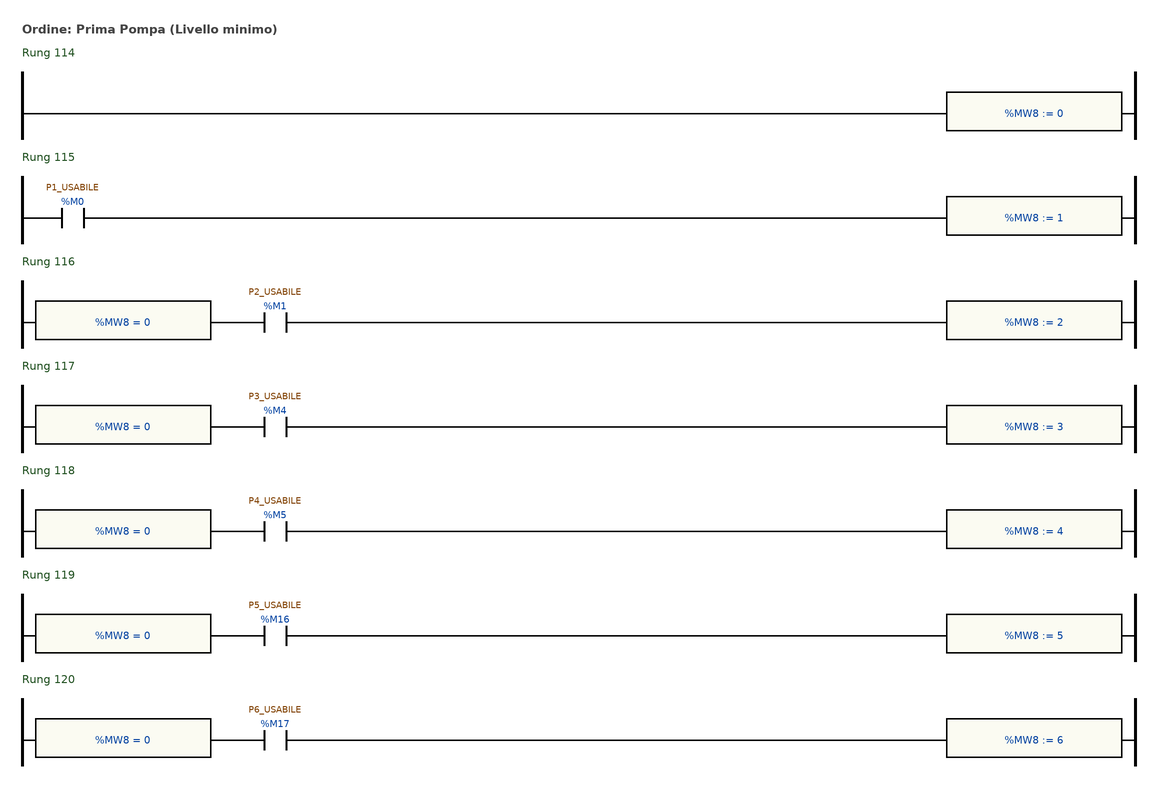

// Rung 114
  LD 1
  [ %MW8 := 0 ]           (* ORDINE_PRIMA_POMPA *)
  // as ST:
  //   ORDINE_PRIMA_POMPA := 0;

// Rung 115
  LD %M0                  (* P1_USABILE *)
  [ %MW8 := 1 ]           (* ORDINE_PRIMA_POMPA *)
  // as ST:
  //   IF P1_USABILE THEN ORDINE_PRIMA_POMPA := 1; END_IF;

// Rung 116
  LD [ %MW8 = 0 ]         (* ORDINE_PRIMA_POMPA *)
  AND %M1                 (* P2_USABILE *)
  [ %MW8 := 2 ]           (* ORDINE_PRIMA_POMPA *)
  // as ST:
  //   IF ORDINE_PRIMA_POMPA = 0 AND P2_USABILE THEN ORDINE_PRIMA_POMPA := 2; END_IF;

// Rung 117
  LD [ %MW8 = 0 ]         (* ORDINE_PRIMA_POMPA *)
  AND %M4                 (* P3_USABILE *)
  [ %MW8 := 3 ]           (* ORDINE_PRIMA_POMPA *)
  // as ST:
  //   IF ORDINE_PRIMA_POMPA = 0 AND P3_USABILE THEN ORDINE_PRIMA_POMPA := 3; END_IF;

// Rung 118
  LD [ %MW8 = 0 ]         (* ORDINE_PRIMA_POMPA *)
  AND %M5                 (* P4_USABILE *)
  [ %MW8 := 4 ]           (* ORDINE_PRIMA_POMPA *)
  // as ST:
  //   IF ORDINE_PRIMA_POMPA = 0 AND P4_USABILE THEN ORDINE_PRIMA_POMPA := 4; END_IF;

// Rung 119
  LD [ %MW8 = 0 ]         (* ORDINE_PRIMA_POMPA *)
  AND %M16                (* P5_USABILE *)
  [ %MW8 := 5 ]           (* ORDINE_PRIMA_POMPA *)
  // as ST:
  //   IF ORDINE_PRIMA_POMPA = 0 AND P5_USABILE THEN ORDINE_PRIMA_POMPA := 5; END_IF;

// Rung 120
  LD [ %MW8 = 0 ]         (* ORDINE_PRIMA_POMPA *)
  AND %M17                (* P6_USABILE *)
  [ %MW8 := 6 ]           (* ORDINE_PRIMA_POMPA *)
  // as ST:
  //   IF ORDINE_PRIMA_POMPA = 0 AND P6_USABILE THEN ORDINE_PRIMA_POMPA := 6; END_IF;

Subroutine Ordine: Seconda Pompa (Livello minimo)
  (* SectionNumber=17, Number=15 *)

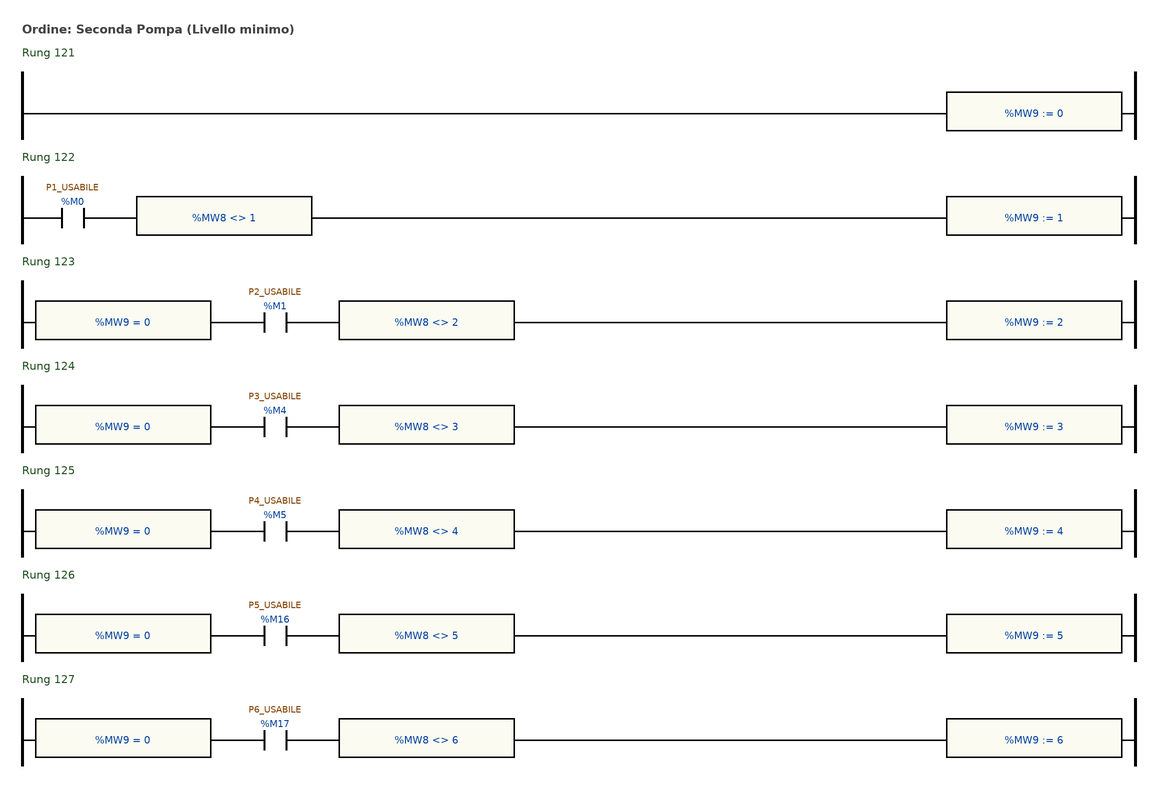

// Rung 121
  LD 1
  [ %MW9 := 0 ]           (* ORDINE_SECONDA_POMPA *)
  // as ST:
  //   ORDINE_SECONDA_POMPA := 0;

// Rung 122
  LD %M0                  (* P1_USABILE *)
  AND [ %MW8 <> 1 ]       (* ORDINE_PRIMA_POMPA *)
  [ %MW9 := 1 ]           (* ORDINE_SECONDA_POMPA *)
  // as ST:
  //   IF P1_USABILE AND ORDINE_PRIMA_POMPA <> 1 THEN ORDINE_SECONDA_POMPA := 1; END_IF;

// Rung 123
  LD [ %MW9 = 0 ]         (* ORDINE_SECONDA_POMPA *)
  AND %M1                 (* P2_USABILE *)
  AND [ %MW8 <> 2 ]       (* ORDINE_PRIMA_POMPA *)
  [ %MW9 := 2 ]           (* ORDINE_SECONDA_POMPA *)
  // as ST:
  //   IF ORDINE_SECONDA_POMPA = 0 AND P2_USABILE AND ORDINE_PRIMA_POMPA <> 2 THEN ORDINE_SECONDA_POMPA := 2; END_IF;

// Rung 124
  LD [ %MW9 = 0 ]         (* ORDINE_SECONDA_POMPA *)
  AND %M4                 (* P3_USABILE *)
  AND [ %MW8 <> 3 ]       (* ORDINE_PRIMA_POMPA *)
  [ %MW9 := 3 ]           (* ORDINE_SECONDA_POMPA *)
  // as ST:
  //   IF ORDINE_SECONDA_POMPA = 0 AND P3_USABILE AND ORDINE_PRIMA_POMPA <> 3 THEN ORDINE_SECONDA_POMPA := 3; END_IF;

// Rung 125
  LD [ %MW9 = 0 ]         (* ORDINE_SECONDA_POMPA *)
  AND %M5                 (* P4_USABILE *)
  AND [ %MW8 <> 4 ]       (* ORDINE_PRIMA_POMPA *)
  [ %MW9 := 4 ]           (* ORDINE_SECONDA_POMPA *)
  // as ST:
  //   IF ORDINE_SECONDA_POMPA = 0 AND P4_USABILE AND ORDINE_PRIMA_POMPA <> 4 THEN ORDINE_SECONDA_POMPA := 4; END_IF;

// Rung 126
  LD [ %MW9 = 0 ]         (* ORDINE_SECONDA_POMPA *)
  AND %M16                (* P5_USABILE *)
  AND [ %MW8 <> 5 ]       (* ORDINE_PRIMA_POMPA *)
  [ %MW9 := 5 ]           (* ORDINE_SECONDA_POMPA *)
  // as ST:
  //   IF ORDINE_SECONDA_POMPA = 0 AND P5_USABILE AND ORDINE_PRIMA_POMPA <> 5 THEN ORDINE_SECONDA_POMPA := 5; END_IF;

// Rung 127
  LD [ %MW9 = 0 ]         (* ORDINE_SECONDA_POMPA *)
  AND %M17                (* P6_USABILE *)
  AND [ %MW8 <> 6 ]       (* ORDINE_PRIMA_POMPA *)
  [ %MW9 := 6 ]           (* ORDINE_SECONDA_POMPA *)
  // as ST:
  //   IF ORDINE_SECONDA_POMPA = 0 AND P6_USABILE AND ORDINE_PRIMA_POMPA <> 6 THEN ORDINE_SECONDA_POMPA := 6; END_IF;

Subroutine Comanda: Prima Pompa (Livello minimo)
  (* SectionNumber=18, Number=16 *)

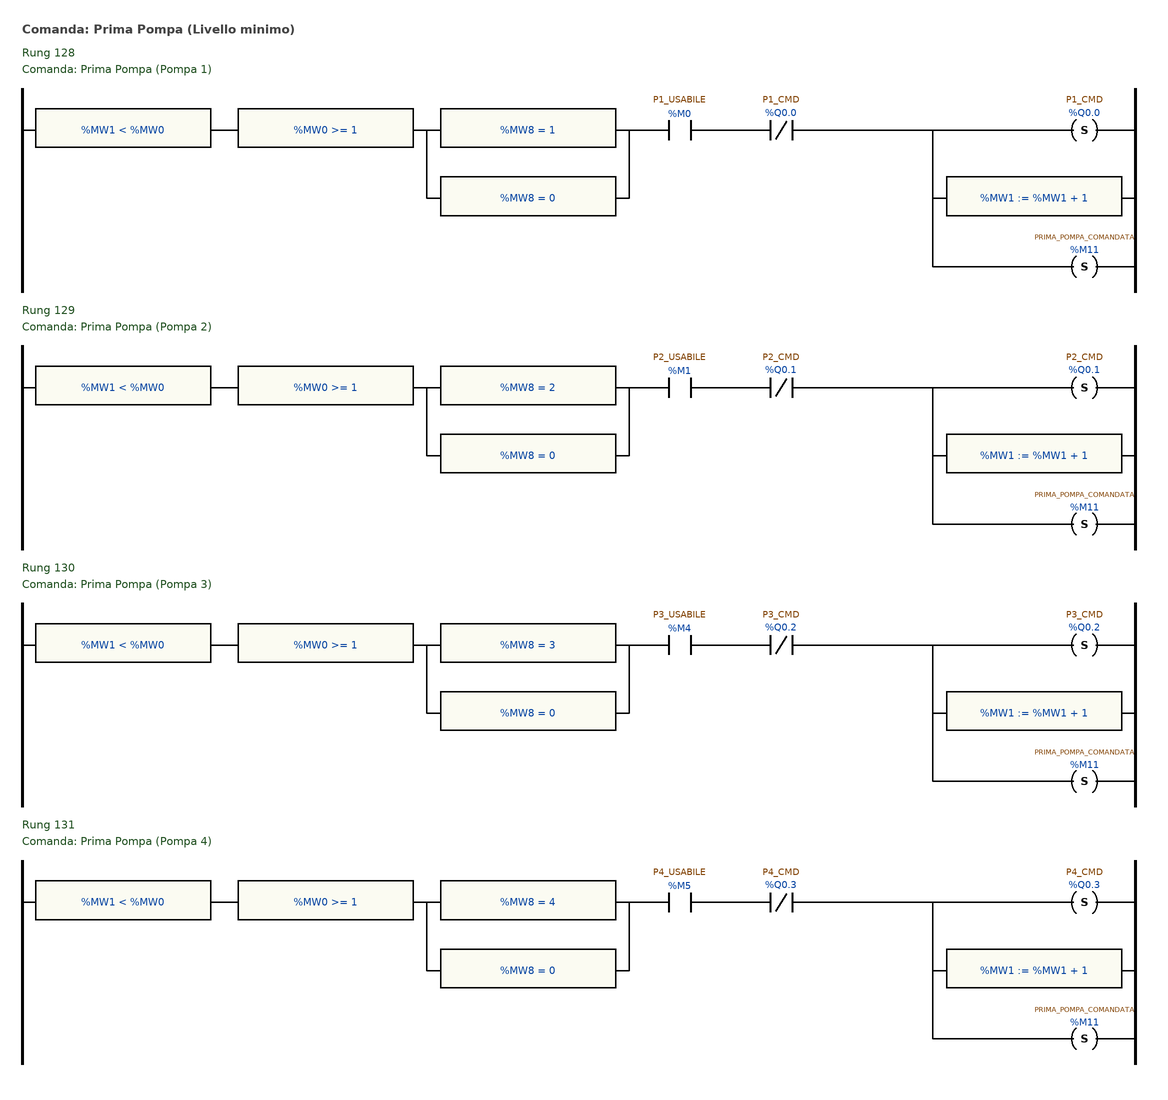

// Rung 128
// Comanda: Prima Pompa (Pompa 1)
  LD [ %MW1 < %MW0 ]      (* NUM_POMPE_COMANDATE, NUM_POMPE_DA_COMANDARE *)
  AND [ %MW0 >= 1 ]       (* NUM_POMPE_DA_COMANDARE *)
  AND( [ %MW8 = 1 ]       (* ORDINE_PRIMA_POMPA *)
  OR [ %MW8 = 0 ]         (* ORDINE_PRIMA_POMPA *)
  )
  AND %M0                 (* P1_USABILE *)
  ANDN %Q0.0              (* P1_CMD *)
  S %Q0.0                 (* P1_CMD *)
  [ %MW1 := %MW1 + 1 ]    (* NUM_POMPE_COMANDATE, NUM_POMPE_COMANDATE *)
  S %M11                  (* PRIMA_POMPA_COMANDATA *)
  // as ST:
  //   _t1 := NUM_POMPE_COMANDATE < NUM_POMPE_DA_COMANDARE AND NUM_POMPE_DA_COMANDARE >= 1 AND (ORDINE_PRIMA_POMPA = 1 OR ORDINE_PRIMA_POMPA = 0) AND P1_USABILE AND NOT P1_CMD;
  //   IF _t1 THEN P1_CMD := TRUE; END_IF;
  //   IF _t1 THEN NUM_POMPE_COMANDATE := NUM_POMPE_COMANDATE + 1; END_IF;
  //   IF _t1 THEN PRIMA_POMPA_COMANDATA := TRUE; END_IF;

// Rung 129
// Comanda: Prima Pompa (Pompa 2)
  LD [ %MW1 < %MW0 ]      (* NUM_POMPE_COMANDATE, NUM_POMPE_DA_COMANDARE *)
  AND [ %MW0 >= 1 ]       (* NUM_POMPE_DA_COMANDARE *)
  AND( [ %MW8 = 2 ]       (* ORDINE_PRIMA_POMPA *)
  OR [ %MW8 = 0 ]         (* ORDINE_PRIMA_POMPA *)
  )
  AND %M1                 (* P2_USABILE *)
  ANDN %Q0.1              (* P2_CMD *)
  S %Q0.1                 (* P2_CMD *)
  [ %MW1 := %MW1 + 1 ]    (* NUM_POMPE_COMANDATE, NUM_POMPE_COMANDATE *)
  S %M11                  (* PRIMA_POMPA_COMANDATA *)
  // as ST:
  //   _t1 := NUM_POMPE_COMANDATE < NUM_POMPE_DA_COMANDARE AND NUM_POMPE_DA_COMANDARE >= 1 AND (ORDINE_PRIMA_POMPA = 2 OR ORDINE_PRIMA_POMPA = 0) AND P2_USABILE AND NOT P2_CMD;
  //   IF _t1 THEN P2_CMD := TRUE; END_IF;
  //   IF _t1 THEN NUM_POMPE_COMANDATE := NUM_POMPE_COMANDATE + 1; END_IF;
  //   IF _t1 THEN PRIMA_POMPA_COMANDATA := TRUE; END_IF;

// Rung 130
// Comanda: Prima Pompa (Pompa 3)
  LD [ %MW1 < %MW0 ]      (* NUM_POMPE_COMANDATE, NUM_POMPE_DA_COMANDARE *)
  AND [ %MW0 >= 1 ]       (* NUM_POMPE_DA_COMANDARE *)
  AND( [ %MW8 = 3 ]       (* ORDINE_PRIMA_POMPA *)
  OR [ %MW8 = 0 ]         (* ORDINE_PRIMA_POMPA *)
  )
  AND %M4                 (* P3_USABILE *)
  ANDN %Q0.2              (* P3_CMD *)
  S %Q0.2                 (* P3_CMD *)
  [ %MW1 := %MW1 + 1 ]    (* NUM_POMPE_COMANDATE, NUM_POMPE_COMANDATE *)
  S %M11                  (* PRIMA_POMPA_COMANDATA *)
  // as ST:
  //   _t1 := NUM_POMPE_COMANDATE < NUM_POMPE_DA_COMANDARE AND NUM_POMPE_DA_COMANDARE >= 1 AND (ORDINE_PRIMA_POMPA = 3 OR ORDINE_PRIMA_POMPA = 0) AND P3_USABILE AND NOT P3_CMD;
  //   IF _t1 THEN P3_CMD := TRUE; END_IF;
  //   IF _t1 THEN NUM_POMPE_COMANDATE := NUM_POMPE_COMANDATE + 1; END_IF;
  //   IF _t1 THEN PRIMA_POMPA_COMANDATA := TRUE; END_IF;

// Rung 131
// Comanda: Prima Pompa (Pompa 4)
  LD [ %MW1 < %MW0 ]      (* NUM_POMPE_COMANDATE, NUM_POMPE_DA_COMANDARE *)
  AND [ %MW0 >= 1 ]       (* NUM_POMPE_DA_COMANDARE *)
  AND( [ %MW8 = 4 ]       (* ORDINE_PRIMA_POMPA *)
  OR [ %MW8 = 0 ]         (* ORDINE_PRIMA_POMPA *)
  )
  AND %M5                 (* P4_USABILE *)
  ANDN %Q0.3              (* P4_CMD *)
  S %Q0.3                 (* P4_CMD *)
  [ %MW1 := %MW1 + 1 ]    (* NUM_POMPE_COMANDATE, NUM_POMPE_COMANDATE *)
  S %M11                  (* PRIMA_POMPA_COMANDATA *)
  // as ST:
  //   _t1 := NUM_POMPE_COMANDATE < NUM_POMPE_DA_COMANDARE AND NUM_POMPE_DA_COMANDARE >= 1 AND (ORDINE_PRIMA_POMPA = 4 OR ORDINE_PRIMA_POMPA = 0) AND P4_USABILE AND NOT P4_CMD;
  //   IF _t1 THEN P4_CMD := TRUE; END_IF;
  //   IF _t1 THEN NUM_POMPE_COMANDATE := NUM_POMPE_COMANDATE + 1; END_IF;
  //   IF _t1 THEN PRIMA_POMPA_COMANDATA := TRUE; END_IF;

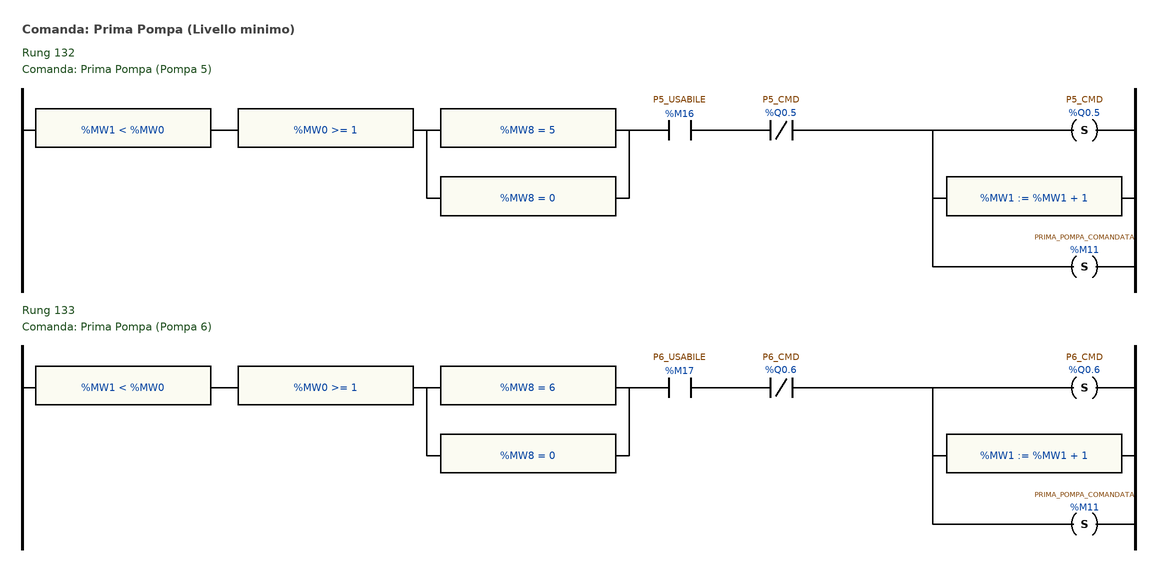

// Rung 132
// Comanda: Prima Pompa (Pompa 5)
  LD [ %MW1 < %MW0 ]      (* NUM_POMPE_COMANDATE, NUM_POMPE_DA_COMANDARE *)
  AND [ %MW0 >= 1 ]       (* NUM_POMPE_DA_COMANDARE *)
  AND( [ %MW8 = 5 ]       (* ORDINE_PRIMA_POMPA *)
  OR [ %MW8 = 0 ]         (* ORDINE_PRIMA_POMPA *)
  )
  AND %M16                (* P5_USABILE *)
  ANDN %Q0.5              (* P5_CMD *)
  S %Q0.5                 (* P5_CMD *)
  [ %MW1 := %MW1 + 1 ]    (* NUM_POMPE_COMANDATE, NUM_POMPE_COMANDATE *)
  S %M11                  (* PRIMA_POMPA_COMANDATA *)
  // as ST:
  //   _t1 := NUM_POMPE_COMANDATE < NUM_POMPE_DA_COMANDARE AND NUM_POMPE_DA_COMANDARE >= 1 AND (ORDINE_PRIMA_POMPA = 5 OR ORDINE_PRIMA_POMPA = 0) AND P5_USABILE AND NOT P5_CMD;
  //   IF _t1 THEN P5_CMD := TRUE; END_IF;
  //   IF _t1 THEN NUM_POMPE_COMANDATE := NUM_POMPE_COMANDATE + 1; END_IF;
  //   IF _t1 THEN PRIMA_POMPA_COMANDATA := TRUE; END_IF;

// Rung 133
// Comanda: Prima Pompa (Pompa 6)
  LD [ %MW1 < %MW0 ]      (* NUM_POMPE_COMANDATE, NUM_POMPE_DA_COMANDARE *)
  AND [ %MW0 >= 1 ]       (* NUM_POMPE_DA_COMANDARE *)
  AND( [ %MW8 = 6 ]       (* ORDINE_PRIMA_POMPA *)
  OR [ %MW8 = 0 ]         (* ORDINE_PRIMA_POMPA *)
  )
  AND %M17                (* P6_USABILE *)
  ANDN %Q0.6              (* P6_CMD *)
  S %Q0.6                 (* P6_CMD *)
  [ %MW1 := %MW1 + 1 ]    (* NUM_POMPE_COMANDATE, NUM_POMPE_COMANDATE *)
  S %M11                  (* PRIMA_POMPA_COMANDATA *)
  // as ST:
  //   _t1 := NUM_POMPE_COMANDATE < NUM_POMPE_DA_COMANDARE AND NUM_POMPE_DA_COMANDARE >= 1 AND (ORDINE_PRIMA_POMPA = 6 OR ORDINE_PRIMA_POMPA = 0) AND P6_USABILE AND NOT P6_CMD;
  //   IF _t1 THEN P6_CMD := TRUE; END_IF;
  //   IF _t1 THEN NUM_POMPE_COMANDATE := NUM_POMPE_COMANDATE + 1; END_IF;
  //   IF _t1 THEN PRIMA_POMPA_COMANDATA := TRUE; END_IF;

Subroutine Comanda: Seconda Pompa (Livello minimo)
  (* SectionNumber=19, Number=17 *)

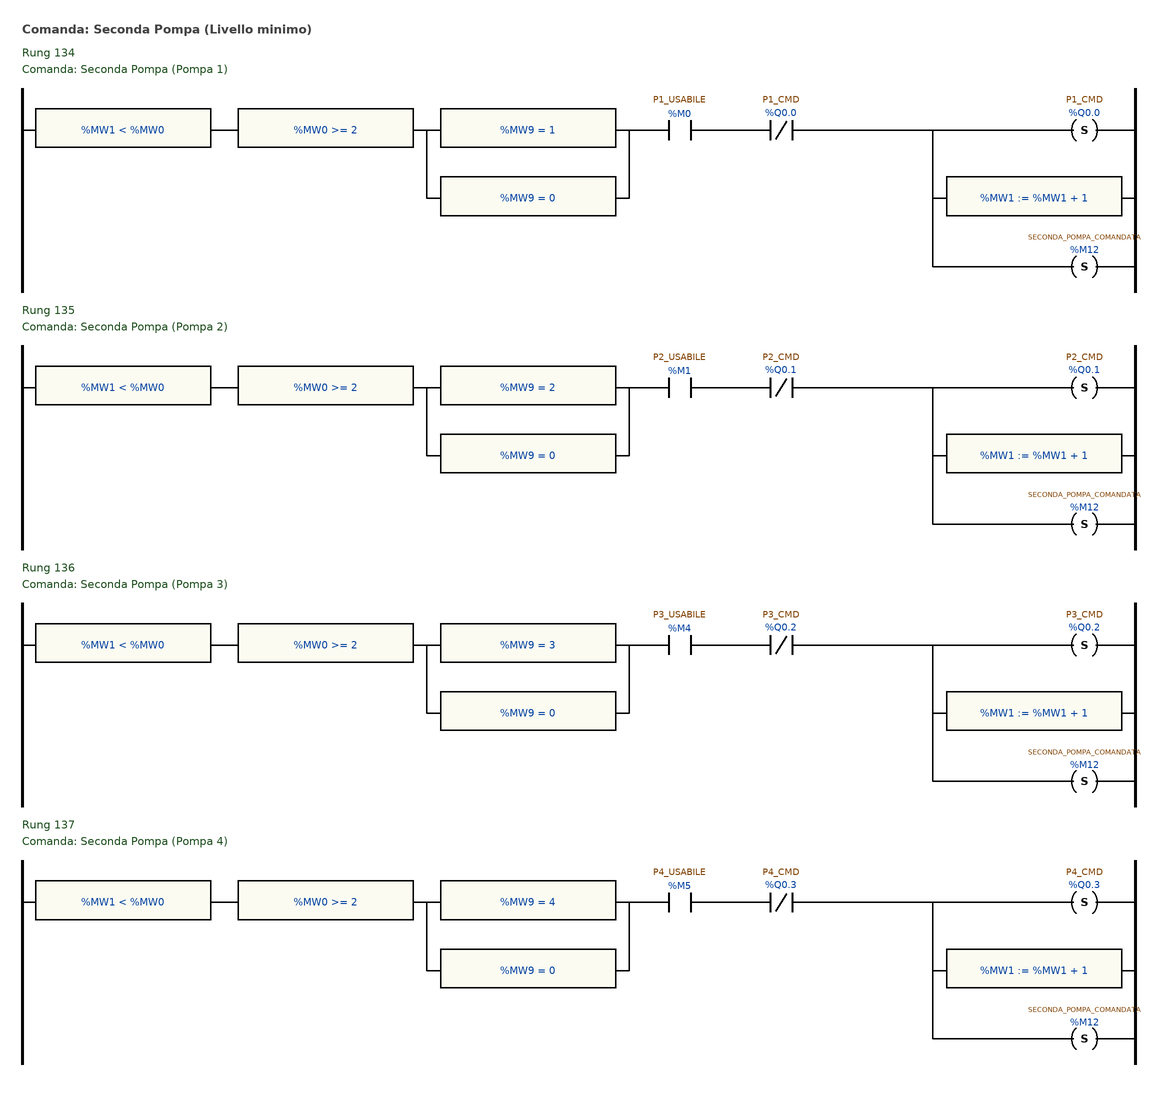

// Rung 134
// Comanda: Seconda Pompa (Pompa 1)
  LD [ %MW1 < %MW0 ]      (* NUM_POMPE_COMANDATE, NUM_POMPE_DA_COMANDARE *)
  AND [ %MW0 >= 2 ]       (* NUM_POMPE_DA_COMANDARE *)
  AND( [ %MW9 = 1 ]       (* ORDINE_SECONDA_POMPA *)
  OR [ %MW9 = 0 ]         (* ORDINE_SECONDA_POMPA *)
  )
  AND %M0                 (* P1_USABILE *)
  ANDN %Q0.0              (* P1_CMD *)
  S %Q0.0                 (* P1_CMD *)
  [ %MW1 := %MW1 + 1 ]    (* NUM_POMPE_COMANDATE, NUM_POMPE_COMANDATE *)
  S %M12                  (* SECONDA_POMPA_COMANDATA *)
  // as ST:
  //   _t1 := NUM_POMPE_COMANDATE < NUM_POMPE_DA_COMANDARE AND NUM_POMPE_DA_COMANDARE >= 2 AND (ORDINE_SECONDA_POMPA = 1 OR ORDINE_SECONDA_POMPA = 0) AND P1_USABILE AND NOT P1_CMD;
  //   IF _t1 THEN P1_CMD := TRUE; END_IF;
  //   IF _t1 THEN NUM_POMPE_COMANDATE := NUM_POMPE_COMANDATE + 1; END_IF;
  //   IF _t1 THEN SECONDA_POMPA_COMANDATA := TRUE; END_IF;

// Rung 135
// Comanda: Seconda Pompa (Pompa 2)
  LD [ %MW1 < %MW0 ]      (* NUM_POMPE_COMANDATE, NUM_POMPE_DA_COMANDARE *)
  AND [ %MW0 >= 2 ]       (* NUM_POMPE_DA_COMANDARE *)
  AND( [ %MW9 = 2 ]       (* ORDINE_SECONDA_POMPA *)
  OR [ %MW9 = 0 ]         (* ORDINE_SECONDA_POMPA *)
  )
  AND %M1                 (* P2_USABILE *)
  ANDN %Q0.1              (* P2_CMD *)
  S %Q0.1                 (* P2_CMD *)
  [ %MW1 := %MW1 + 1 ]    (* NUM_POMPE_COMANDATE, NUM_POMPE_COMANDATE *)
  S %M12                  (* SECONDA_POMPA_COMANDATA *)
  // as ST:
  //   _t1 := NUM_POMPE_COMANDATE < NUM_POMPE_DA_COMANDARE AND NUM_POMPE_DA_COMANDARE >= 2 AND (ORDINE_SECONDA_POMPA = 2 OR ORDINE_SECONDA_POMPA = 0) AND P2_USABILE AND NOT P2_CMD;
  //   IF _t1 THEN P2_CMD := TRUE; END_IF;
  //   IF _t1 THEN NUM_POMPE_COMANDATE := NUM_POMPE_COMANDATE + 1; END_IF;
  //   IF _t1 THEN SECONDA_POMPA_COMANDATA := TRUE; END_IF;

// Rung 136
// Comanda: Seconda Pompa (Pompa 3)
  LD [ %MW1 < %MW0 ]      (* NUM_POMPE_COMANDATE, NUM_POMPE_DA_COMANDARE *)
  AND [ %MW0 >= 2 ]       (* NUM_POMPE_DA_COMANDARE *)
  AND( [ %MW9 = 3 ]       (* ORDINE_SECONDA_POMPA *)
  OR [ %MW9 = 0 ]         (* ORDINE_SECONDA_POMPA *)
  )
  AND %M4                 (* P3_USABILE *)
  ANDN %Q0.2              (* P3_CMD *)
  S %Q0.2                 (* P3_CMD *)
  [ %MW1 := %MW1 + 1 ]    (* NUM_POMPE_COMANDATE, NUM_POMPE_COMANDATE *)
  S %M12                  (* SECONDA_POMPA_COMANDATA *)
  // as ST:
  //   _t1 := NUM_POMPE_COMANDATE < NUM_POMPE_DA_COMANDARE AND NUM_POMPE_DA_COMANDARE >= 2 AND (ORDINE_SECONDA_POMPA = 3 OR ORDINE_SECONDA_POMPA = 0) AND P3_USABILE AND NOT P3_CMD;
  //   IF _t1 THEN P3_CMD := TRUE; END_IF;
  //   IF _t1 THEN NUM_POMPE_COMANDATE := NUM_POMPE_COMANDATE + 1; END_IF;
  //   IF _t1 THEN SECONDA_POMPA_COMANDATA := TRUE; END_IF;

// Rung 137
// Comanda: Seconda Pompa (Pompa 4)
  LD [ %MW1 < %MW0 ]      (* NUM_POMPE_COMANDATE, NUM_POMPE_DA_COMANDARE *)
  AND [ %MW0 >= 2 ]       (* NUM_POMPE_DA_COMANDARE *)
  AND( [ %MW9 = 4 ]       (* ORDINE_SECONDA_POMPA *)
  OR [ %MW9 = 0 ]         (* ORDINE_SECONDA_POMPA *)
  )
  AND %M5                 (* P4_USABILE *)
  ANDN %Q0.3              (* P4_CMD *)
  S %Q0.3                 (* P4_CMD *)
  [ %MW1 := %MW1 + 1 ]    (* NUM_POMPE_COMANDATE, NUM_POMPE_COMANDATE *)
  S %M12                  (* SECONDA_POMPA_COMANDATA *)
  // as ST:
  //   _t1 := NUM_POMPE_COMANDATE < NUM_POMPE_DA_COMANDARE AND NUM_POMPE_DA_COMANDARE >= 2 AND (ORDINE_SECONDA_POMPA = 4 OR ORDINE_SECONDA_POMPA = 0) AND P4_USABILE AND NOT P4_CMD;
  //   IF _t1 THEN P4_CMD := TRUE; END_IF;
  //   IF _t1 THEN NUM_POMPE_COMANDATE := NUM_POMPE_COMANDATE + 1; END_IF;
  //   IF _t1 THEN SECONDA_POMPA_COMANDATA := TRUE; END_IF;

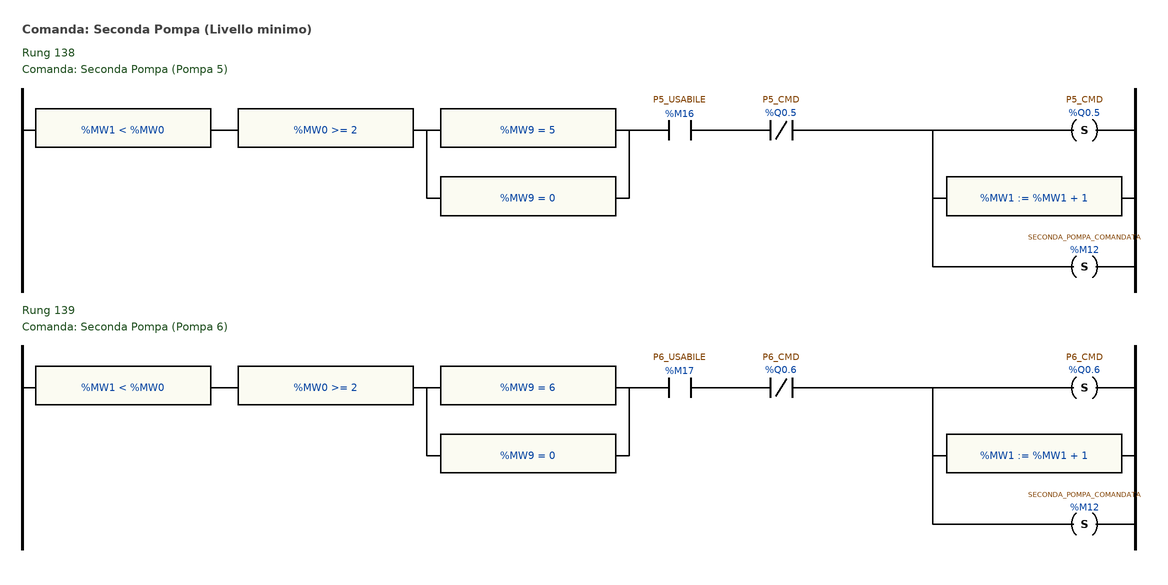

// Rung 138
// Comanda: Seconda Pompa (Pompa 5)
  LD [ %MW1 < %MW0 ]      (* NUM_POMPE_COMANDATE, NUM_POMPE_DA_COMANDARE *)
  AND [ %MW0 >= 2 ]       (* NUM_POMPE_DA_COMANDARE *)
  AND( [ %MW9 = 5 ]       (* ORDINE_SECONDA_POMPA *)
  OR [ %MW9 = 0 ]         (* ORDINE_SECONDA_POMPA *)
  )
  AND %M16                (* P5_USABILE *)
  ANDN %Q0.5              (* P5_CMD *)
  S %Q0.5                 (* P5_CMD *)
  [ %MW1 := %MW1 + 1 ]    (* NUM_POMPE_COMANDATE, NUM_POMPE_COMANDATE *)
  S %M12                  (* SECONDA_POMPA_COMANDATA *)
  // as ST:
  //   _t1 := NUM_POMPE_COMANDATE < NUM_POMPE_DA_COMANDARE AND NUM_POMPE_DA_COMANDARE >= 2 AND (ORDINE_SECONDA_POMPA = 5 OR ORDINE_SECONDA_POMPA = 0) AND P5_USABILE AND NOT P5_CMD;
  //   IF _t1 THEN P5_CMD := TRUE; END_IF;
  //   IF _t1 THEN NUM_POMPE_COMANDATE := NUM_POMPE_COMANDATE + 1; END_IF;
  //   IF _t1 THEN SECONDA_POMPA_COMANDATA := TRUE; END_IF;

// Rung 139
// Comanda: Seconda Pompa (Pompa 6)
  LD [ %MW1 < %MW0 ]      (* NUM_POMPE_COMANDATE, NUM_POMPE_DA_COMANDARE *)
  AND [ %MW0 >= 2 ]       (* NUM_POMPE_DA_COMANDARE *)
  AND( [ %MW9 = 6 ]       (* ORDINE_SECONDA_POMPA *)
  OR [ %MW9 = 0 ]         (* ORDINE_SECONDA_POMPA *)
  )
  AND %M17                (* P6_USABILE *)
  ANDN %Q0.6              (* P6_CMD *)
  S %Q0.6                 (* P6_CMD *)
  [ %MW1 := %MW1 + 1 ]    (* NUM_POMPE_COMANDATE, NUM_POMPE_COMANDATE *)
  S %M12                  (* SECONDA_POMPA_COMANDATA *)
  // as ST:
  //   _t1 := NUM_POMPE_COMANDATE < NUM_POMPE_DA_COMANDARE AND NUM_POMPE_DA_COMANDARE >= 2 AND (ORDINE_SECONDA_POMPA = 6 OR ORDINE_SECONDA_POMPA = 0) AND P6_USABILE AND NOT P6_CMD;
  //   IF _t1 THEN P6_CMD := TRUE; END_IF;
  //   IF _t1 THEN NUM_POMPE_COMANDATE := NUM_POMPE_COMANDATE + 1; END_IF;
  //   IF _t1 THEN SECONDA_POMPA_COMANDATA := TRUE; END_IF;

Subroutine Disattivazione Pompe (Livello minimo)
  (* SectionNumber=20, Number=18 *)

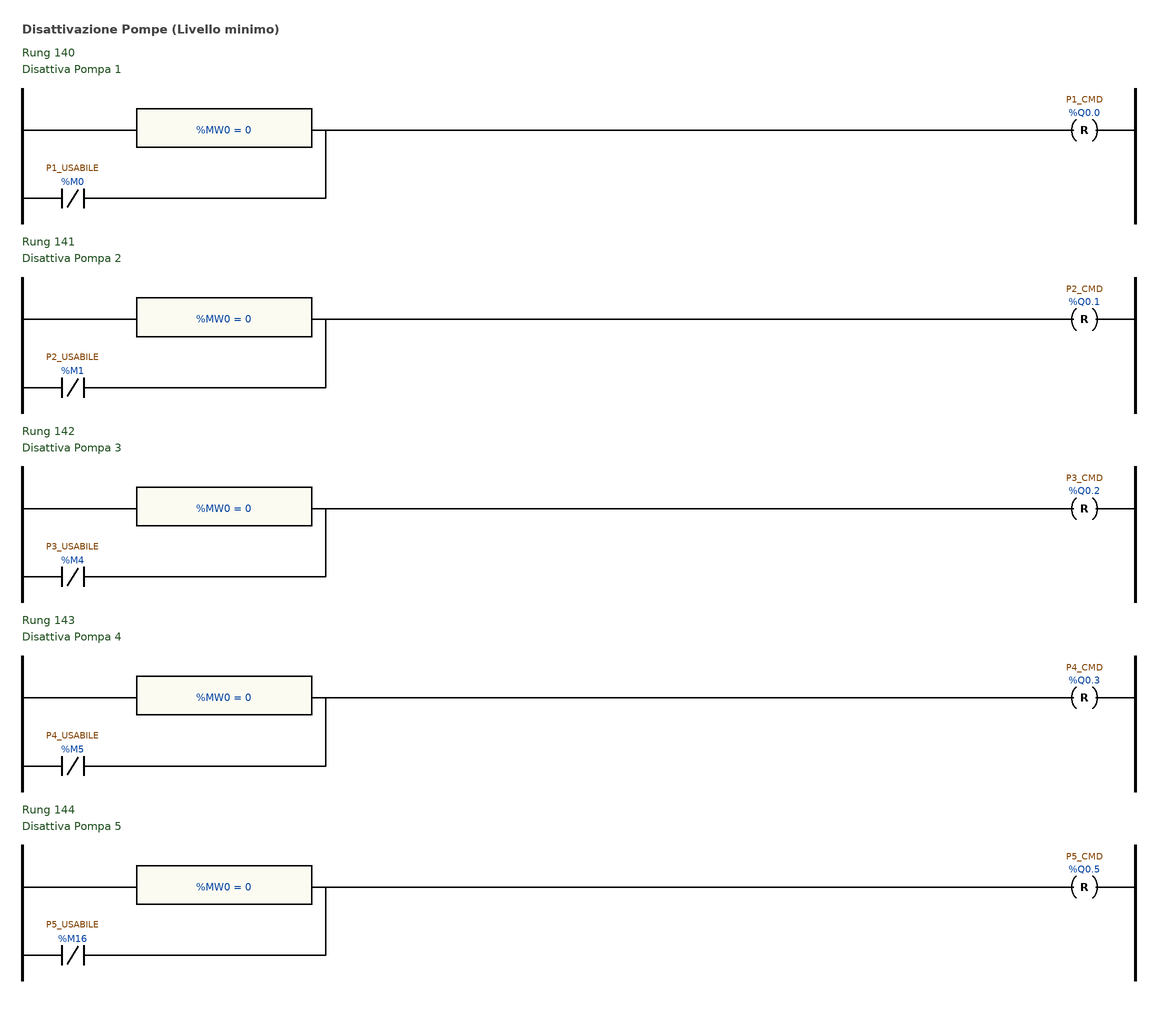

// Rung 140
// Disattiva Pompa 1
  LD [ %MW0 = 0 ]         (* NUM_POMPE_DA_COMANDARE *)
  ORN %M0                 (* P1_USABILE *)
  R %Q0.0                 (* P1_CMD *)
  // as ST:
  //   IF NUM_POMPE_DA_COMANDARE = 0 OR NOT P1_USABILE THEN P1_CMD := FALSE; END_IF;

// Rung 141
// Disattiva Pompa 2
  LD [ %MW0 = 0 ]         (* NUM_POMPE_DA_COMANDARE *)
  ORN %M1                 (* P2_USABILE *)
  R %Q0.1                 (* P2_CMD *)
  // as ST:
  //   IF NUM_POMPE_DA_COMANDARE = 0 OR NOT P2_USABILE THEN P2_CMD := FALSE; END_IF;

// Rung 142
// Disattiva Pompa 3
  LD [ %MW0 = 0 ]         (* NUM_POMPE_DA_COMANDARE *)
  ORN %M4                 (* P3_USABILE *)
  R %Q0.2                 (* P3_CMD *)
  // as ST:
  //   IF NUM_POMPE_DA_COMANDARE = 0 OR NOT P3_USABILE THEN P3_CMD := FALSE; END_IF;

// Rung 143
// Disattiva Pompa 4
  LD [ %MW0 = 0 ]         (* NUM_POMPE_DA_COMANDARE *)
  ORN %M5                 (* P4_USABILE *)
  R %Q0.3                 (* P4_CMD *)
  // as ST:
  //   IF NUM_POMPE_DA_COMANDARE = 0 OR NOT P4_USABILE THEN P4_CMD := FALSE; END_IF;

// Rung 144
// Disattiva Pompa 5
  LD [ %MW0 = 0 ]         (* NUM_POMPE_DA_COMANDARE *)
  ORN %M16                (* P5_USABILE *)
  R %Q0.5                 (* P5_CMD *)
  // as ST:
  //   IF NUM_POMPE_DA_COMANDARE = 0 OR NOT P5_USABILE THEN P5_CMD := FALSE; END_IF;

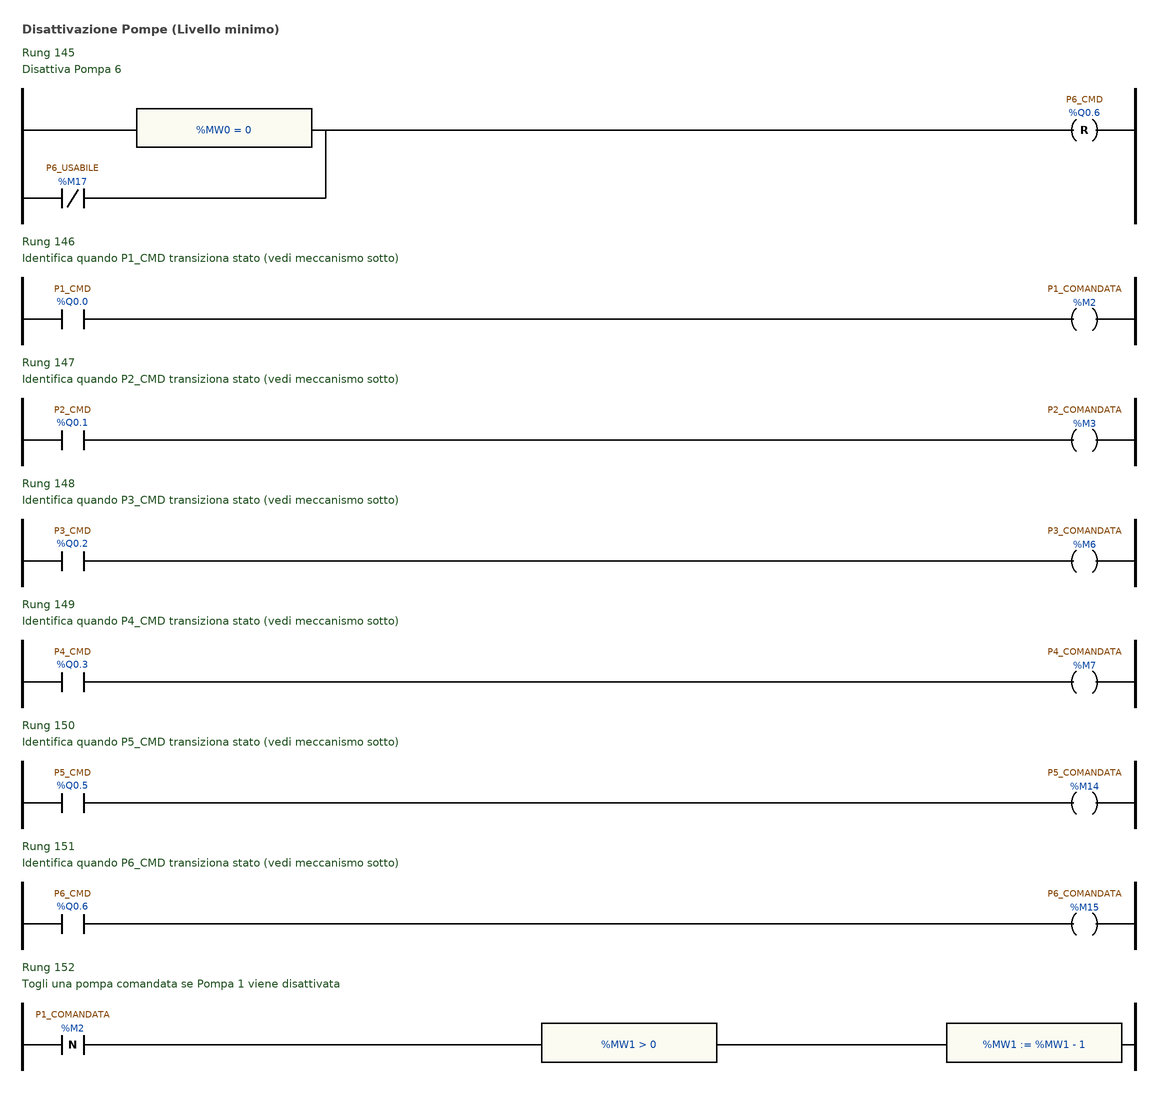

// Rung 145
// Disattiva Pompa 6
  LD [ %MW0 = 0 ]         (* NUM_POMPE_DA_COMANDARE *)
  ORN %M17                (* P6_USABILE *)
  R %Q0.6                 (* P6_CMD *)
  // as ST:
  //   IF NUM_POMPE_DA_COMANDARE = 0 OR NOT P6_USABILE THEN P6_CMD := FALSE; END_IF;

// Rung 146
// Identifica quando P1_CMD transiziona stato (vedi meccanismo sotto)
  LD %Q0.0                (* P1_CMD *)
  ST %M2                  (* P1_COMANDATA *)
  // as ST:
  //   P1_COMANDATA := P1_CMD;

// Rung 147
// Identifica quando P2_CMD transiziona stato (vedi meccanismo sotto)
  LD %Q0.1                (* P2_CMD *)
  ST %M3                  (* P2_COMANDATA *)
  // as ST:
  //   P2_COMANDATA := P2_CMD;

// Rung 148
// Identifica quando P3_CMD transiziona stato (vedi meccanismo sotto)
  LD %Q0.2                (* P3_CMD *)
  ST %M6                  (* P3_COMANDATA *)
  // as ST:
  //   P3_COMANDATA := P3_CMD;

// Rung 149
// Identifica quando P4_CMD transiziona stato (vedi meccanismo sotto)
  LD %Q0.3                (* P4_CMD *)
  ST %M7                  (* P4_COMANDATA *)
  // as ST:
  //   P4_COMANDATA := P4_CMD;

// Rung 150
// Identifica quando P5_CMD transiziona stato (vedi meccanismo sotto)
  LD %Q0.5                (* P5_CMD *)
  ST %M14                 (* P5_COMANDATA *)
  // as ST:
  //   P5_COMANDATA := P5_CMD;

// Rung 151
// Identifica quando P6_CMD transiziona stato (vedi meccanismo sotto)
  LD %Q0.6                (* P6_CMD *)
  ST %M15                 (* P6_COMANDATA *)
  // as ST:
  //   P6_COMANDATA := P6_CMD;

// Rung 152
// Togli una pompa comandata se Pompa 1 viene disattivata
  LDF %M2                 (* P1_COMANDATA *)
  AND [ %MW1 > 0 ]        (* NUM_POMPE_COMANDATE *)
  [ %MW1 := %MW1 - 1 ]    (* NUM_POMPE_COMANDATE, NUM_POMPE_COMANDATE *)
  // as ST:
  //   IF FALLING(P1_COMANDATA) AND NUM_POMPE_COMANDATE > 0 THEN NUM_POMPE_COMANDATE := NUM_POMPE_COMANDATE - 1; END_IF;

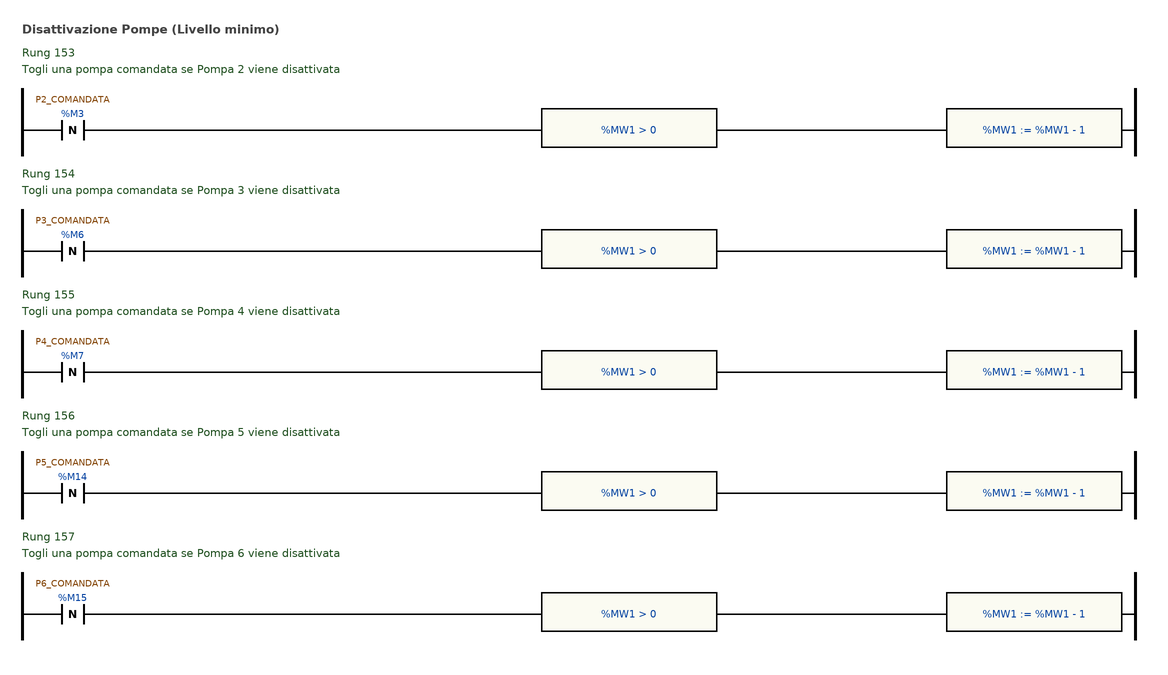

// Rung 153
// Togli una pompa comandata se Pompa 2 viene disattivata
  LDF %M3                 (* P2_COMANDATA *)
  AND [ %MW1 > 0 ]        (* NUM_POMPE_COMANDATE *)
  [ %MW1 := %MW1 - 1 ]    (* NUM_POMPE_COMANDATE, NUM_POMPE_COMANDATE *)
  // as ST:
  //   IF FALLING(P2_COMANDATA) AND NUM_POMPE_COMANDATE > 0 THEN NUM_POMPE_COMANDATE := NUM_POMPE_COMANDATE - 1; END_IF;

// Rung 154
// Togli una pompa comandata se Pompa 3 viene disattivata
  LDF %M6                 (* P3_COMANDATA *)
  AND [ %MW1 > 0 ]        (* NUM_POMPE_COMANDATE *)
  [ %MW1 := %MW1 - 1 ]    (* NUM_POMPE_COMANDATE, NUM_POMPE_COMANDATE *)
  // as ST:
  //   IF FALLING(P3_COMANDATA) AND NUM_POMPE_COMANDATE > 0 THEN NUM_POMPE_COMANDATE := NUM_POMPE_COMANDATE - 1; END_IF;

// Rung 155
// Togli una pompa comandata se Pompa 4 viene disattivata
  LDF %M7                 (* P4_COMANDATA *)
  AND [ %MW1 > 0 ]        (* NUM_POMPE_COMANDATE *)
  [ %MW1 := %MW1 - 1 ]    (* NUM_POMPE_COMANDATE, NUM_POMPE_COMANDATE *)
  // as ST:
  //   IF FALLING(P4_COMANDATA) AND NUM_POMPE_COMANDATE > 0 THEN NUM_POMPE_COMANDATE := NUM_POMPE_COMANDATE - 1; END_IF;

// Rung 156
// Togli una pompa comandata se Pompa 5 viene disattivata
  LDF %M14                (* P5_COMANDATA *)
  AND [ %MW1 > 0 ]        (* NUM_POMPE_COMANDATE *)
  [ %MW1 := %MW1 - 1 ]    (* NUM_POMPE_COMANDATE, NUM_POMPE_COMANDATE *)
  // as ST:
  //   IF FALLING(P5_COMANDATA) AND NUM_POMPE_COMANDATE > 0 THEN NUM_POMPE_COMANDATE := NUM_POMPE_COMANDATE - 1; END_IF;

// Rung 157
// Togli una pompa comandata se Pompa 6 viene disattivata
  LDF %M15                (* P6_COMANDATA *)
  AND [ %MW1 > 0 ]        (* NUM_POMPE_COMANDATE *)
  [ %MW1 := %MW1 - 1 ]    (* NUM_POMPE_COMANDATE, NUM_POMPE_COMANDATE *)
  // as ST:
  //   IF FALLING(P6_COMANDATA) AND NUM_POMPE_COMANDATE > 0 THEN NUM_POMPE_COMANDATE := NUM_POMPE_COMANDATE - 1; END_IF;

Subroutine Soglie (Livello minimo)
  (* SectionNumber=21, Number=19 *)

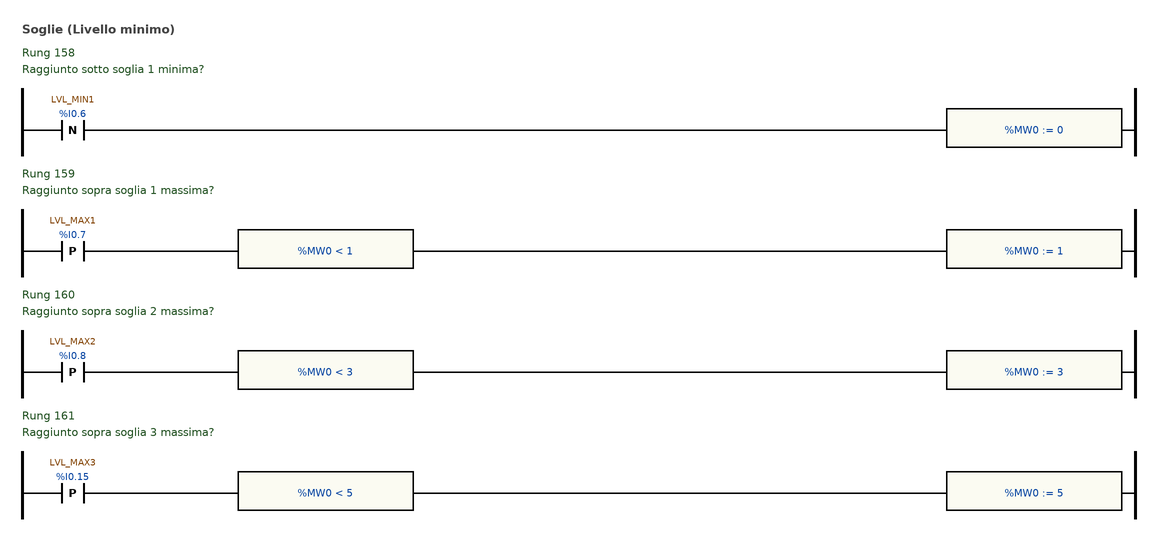

// Rung 158
// Raggiunto sotto soglia 1 minima?
  LDF %I0.6               (* LVL_MIN1 *)
  [ %MW0 := 0 ]           (* NUM_POMPE_DA_COMANDARE *)
  // as ST:
  //   IF FALLING(LVL_MIN1) THEN NUM_POMPE_DA_COMANDARE := 0; END_IF;

// Rung 159
// Raggiunto sopra soglia 1 massima?
  LDR %I0.7               (* LVL_MAX1 *)
  AND [ %MW0 < 1 ]        (* NUM_POMPE_DA_COMANDARE *)
  [ %MW0 := 1 ]           (* NUM_POMPE_DA_COMANDARE *)
  // as ST:
  //   IF RISING(LVL_MAX1) AND NUM_POMPE_DA_COMANDARE < 1 THEN NUM_POMPE_DA_COMANDARE := 1; END_IF;

// Rung 160
// Raggiunto sopra soglia 2 massima?
  LDR %I0.8               (* LVL_MAX2 *)
  AND [ %MW0 < 3 ]        (* NUM_POMPE_DA_COMANDARE *)
  [ %MW0 := 3 ]           (* NUM_POMPE_DA_COMANDARE *)
  // as ST:
  //   IF RISING(LVL_MAX2) AND NUM_POMPE_DA_COMANDARE < 3 THEN NUM_POMPE_DA_COMANDARE := 3; END_IF;

// Rung 161
// Raggiunto sopra soglia 3 massima?
  LDR %I0.15              (* LVL_MAX3 *)
  AND [ %MW0 < 5 ]        (* NUM_POMPE_DA_COMANDARE *)
  [ %MW0 := 5 ]           (* NUM_POMPE_DA_COMANDARE *)
  // as ST:
  //   IF RISING(LVL_MAX3) AND NUM_POMPE_DA_COMANDARE < 5 THEN NUM_POMPE_DA_COMANDARE := 5; END_IF;

Subroutine Ordine: Terza Pompa (Livello minimo)
  (* SectionNumber=22, Number=20 *)

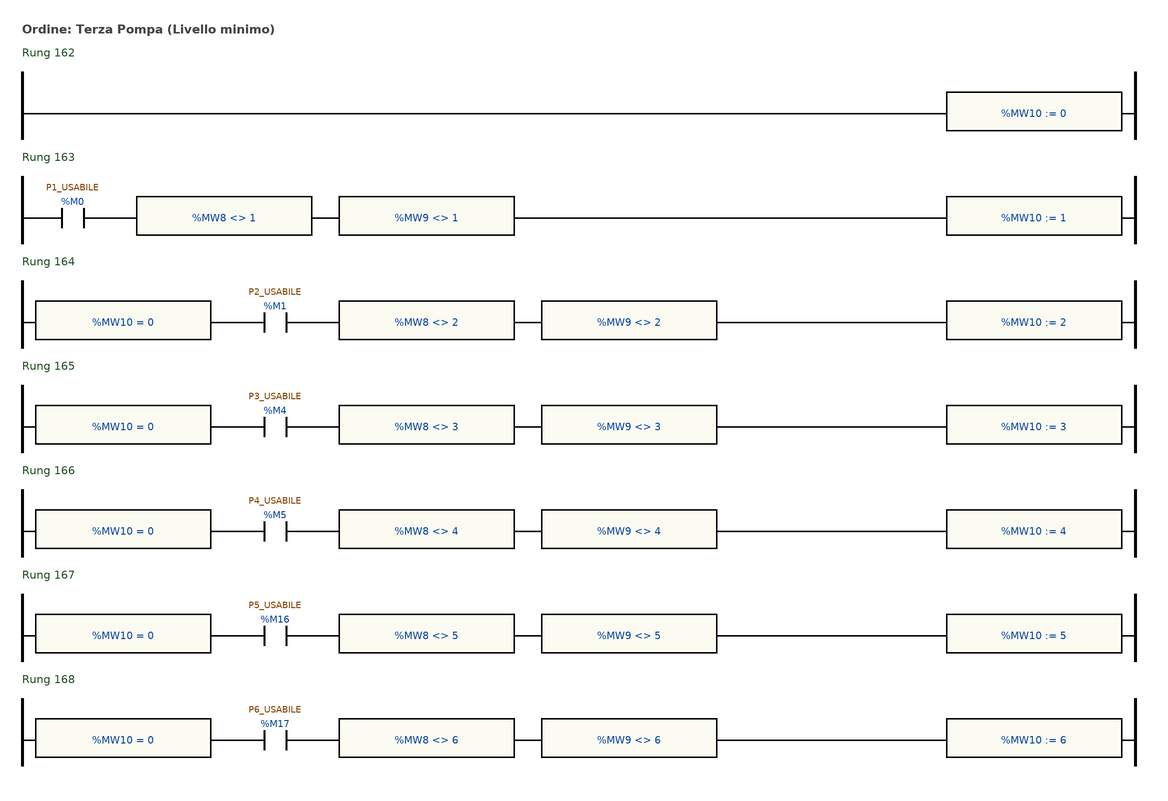

// Rung 162
  LD 1
  [ %MW10 := 0 ]          (* ORDINE_TERZA_POMPA *)
  // as ST:
  //   ORDINE_TERZA_POMPA := 0;

// Rung 163
  LD %M0                  (* P1_USABILE *)
  AND [ %MW8 <> 1 ]       (* ORDINE_PRIMA_POMPA *)
  AND [ %MW9 <> 1 ]       (* ORDINE_SECONDA_POMPA *)
  [ %MW10 := 1 ]          (* ORDINE_TERZA_POMPA *)
  // as ST:
  //   IF P1_USABILE AND ORDINE_PRIMA_POMPA <> 1 AND ORDINE_SECONDA_POMPA <> 1 THEN ORDINE_TERZA_POMPA := 1; END_IF;

// Rung 164
  LD [ %MW10 = 0 ]        (* ORDINE_TERZA_POMPA *)
  AND %M1                 (* P2_USABILE *)
  AND [ %MW8 <> 2 ]       (* ORDINE_PRIMA_POMPA *)
  AND [ %MW9 <> 2 ]       (* ORDINE_SECONDA_POMPA *)
  [ %MW10 := 2 ]          (* ORDINE_TERZA_POMPA *)
  // as ST:
  //   IF ORDINE_TERZA_POMPA = 0 AND P2_USABILE AND ORDINE_PRIMA_POMPA <> 2 AND ORDINE_SECONDA_POMPA <> 2 THEN ORDINE_TERZA_POMPA := 2; END_IF;

// Rung 165
  LD [ %MW10 = 0 ]        (* ORDINE_TERZA_POMPA *)
  AND %M4                 (* P3_USABILE *)
  AND [ %MW8 <> 3 ]       (* ORDINE_PRIMA_POMPA *)
  AND [ %MW9 <> 3 ]       (* ORDINE_SECONDA_POMPA *)
  [ %MW10 := 3 ]          (* ORDINE_TERZA_POMPA *)
  // as ST:
  //   IF ORDINE_TERZA_POMPA = 0 AND P3_USABILE AND ORDINE_PRIMA_POMPA <> 3 AND ORDINE_SECONDA_POMPA <> 3 THEN ORDINE_TERZA_POMPA := 3; END_IF;

// Rung 166
  LD [ %MW10 = 0 ]        (* ORDINE_TERZA_POMPA *)
  AND %M5                 (* P4_USABILE *)
  AND [ %MW8 <> 4 ]       (* ORDINE_PRIMA_POMPA *)
  AND [ %MW9 <> 4 ]       (* ORDINE_SECONDA_POMPA *)
  [ %MW10 := 4 ]          (* ORDINE_TERZA_POMPA *)
  // as ST:
  //   IF ORDINE_TERZA_POMPA = 0 AND P4_USABILE AND ORDINE_PRIMA_POMPA <> 4 AND ORDINE_SECONDA_POMPA <> 4 THEN ORDINE_TERZA_POMPA := 4; END_IF;

// Rung 167
  LD [ %MW10 = 0 ]        (* ORDINE_TERZA_POMPA *)
  AND %M16                (* P5_USABILE *)
  AND [ %MW8 <> 5 ]       (* ORDINE_PRIMA_POMPA *)
  AND [ %MW9 <> 5 ]       (* ORDINE_SECONDA_POMPA *)
  [ %MW10 := 5 ]          (* ORDINE_TERZA_POMPA *)
  // as ST:
  //   IF ORDINE_TERZA_POMPA = 0 AND P5_USABILE AND ORDINE_PRIMA_POMPA <> 5 AND ORDINE_SECONDA_POMPA <> 5 THEN ORDINE_TERZA_POMPA := 5; END_IF;

// Rung 168
  LD [ %MW10 = 0 ]        (* ORDINE_TERZA_POMPA *)
  AND %M17                (* P6_USABILE *)
  AND [ %MW8 <> 6 ]       (* ORDINE_PRIMA_POMPA *)
  AND [ %MW9 <> 6 ]       (* ORDINE_SECONDA_POMPA *)
  [ %MW10 := 6 ]          (* ORDINE_TERZA_POMPA *)
  // as ST:
  //   IF ORDINE_TERZA_POMPA = 0 AND P6_USABILE AND ORDINE_PRIMA_POMPA <> 6 AND ORDINE_SECONDA_POMPA <> 6 THEN ORDINE_TERZA_POMPA := 6; END_IF;

Subroutine Comanda: Terza Pompa (Livello minimo)
  (* SectionNumber=23, Number=21 *)

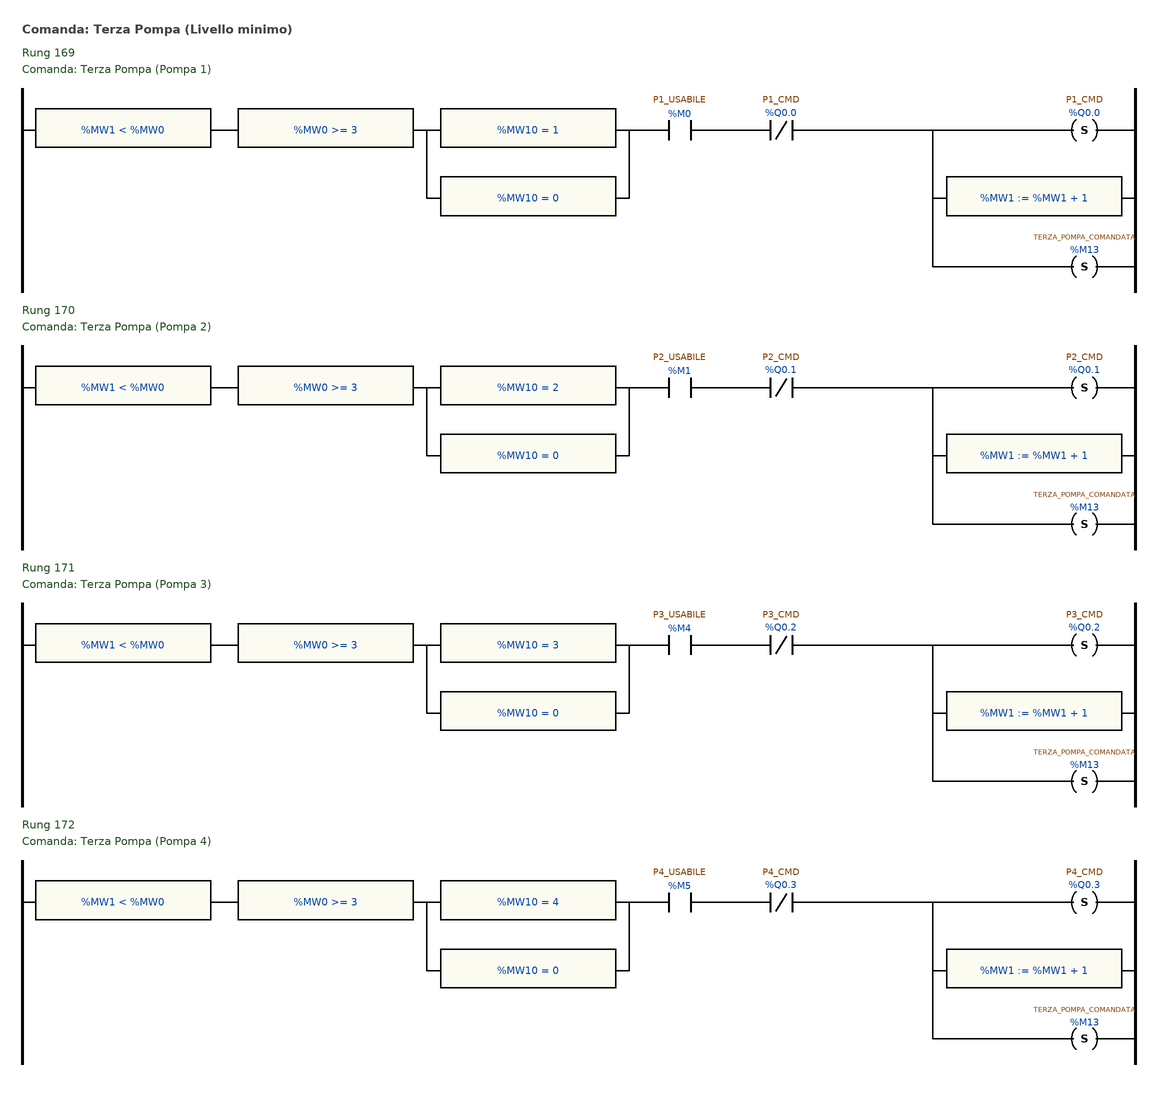

// Rung 169
// Comanda: Terza Pompa (Pompa 1)
  LD [ %MW1 < %MW0 ]      (* NUM_POMPE_COMANDATE, NUM_POMPE_DA_COMANDARE *)
  AND [ %MW0 >= 3 ]       (* NUM_POMPE_DA_COMANDARE *)
  AND( [ %MW10 = 1 ]      (* ORDINE_TERZA_POMPA *)
  OR [ %MW10 = 0 ]        (* ORDINE_TERZA_POMPA *)
  )
  AND %M0                 (* P1_USABILE *)
  ANDN %Q0.0              (* P1_CMD *)
  S %Q0.0                 (* P1_CMD *)
  [ %MW1 := %MW1 + 1 ]    (* NUM_POMPE_COMANDATE, NUM_POMPE_COMANDATE *)
  S %M13                  (* TERZA_POMPA_COMANDATA *)
  // as ST:
  //   _t1 := NUM_POMPE_COMANDATE < NUM_POMPE_DA_COMANDARE AND NUM_POMPE_DA_COMANDARE >= 3 AND (ORDINE_TERZA_POMPA = 1 OR ORDINE_TERZA_POMPA = 0) AND P1_USABILE AND NOT P1_CMD;
  //   IF _t1 THEN P1_CMD := TRUE; END_IF;
  //   IF _t1 THEN NUM_POMPE_COMANDATE := NUM_POMPE_COMANDATE + 1; END_IF;
  //   IF _t1 THEN TERZA_POMPA_COMANDATA := TRUE; END_IF;

// Rung 170
// Comanda: Terza Pompa (Pompa 2)
  LD [ %MW1 < %MW0 ]      (* NUM_POMPE_COMANDATE, NUM_POMPE_DA_COMANDARE *)
  AND [ %MW0 >= 3 ]       (* NUM_POMPE_DA_COMANDARE *)
  AND( [ %MW10 = 2 ]      (* ORDINE_TERZA_POMPA *)
  OR [ %MW10 = 0 ]        (* ORDINE_TERZA_POMPA *)
  )
  AND %M1                 (* P2_USABILE *)
  ANDN %Q0.1              (* P2_CMD *)
  S %Q0.1                 (* P2_CMD *)
  [ %MW1 := %MW1 + 1 ]    (* NUM_POMPE_COMANDATE, NUM_POMPE_COMANDATE *)
  S %M13                  (* TERZA_POMPA_COMANDATA *)
  // as ST:
  //   _t1 := NUM_POMPE_COMANDATE < NUM_POMPE_DA_COMANDARE AND NUM_POMPE_DA_COMANDARE >= 3 AND (ORDINE_TERZA_POMPA = 2 OR ORDINE_TERZA_POMPA = 0) AND P2_USABILE AND NOT P2_CMD;
  //   IF _t1 THEN P2_CMD := TRUE; END_IF;
  //   IF _t1 THEN NUM_POMPE_COMANDATE := NUM_POMPE_COMANDATE + 1; END_IF;
  //   IF _t1 THEN TERZA_POMPA_COMANDATA := TRUE; END_IF;

// Rung 171
// Comanda: Terza Pompa (Pompa 3)
  LD [ %MW1 < %MW0 ]      (* NUM_POMPE_COMANDATE, NUM_POMPE_DA_COMANDARE *)
  AND [ %MW0 >= 3 ]       (* NUM_POMPE_DA_COMANDARE *)
  AND( [ %MW10 = 3 ]      (* ORDINE_TERZA_POMPA *)
  OR [ %MW10 = 0 ]        (* ORDINE_TERZA_POMPA *)
  )
  AND %M4                 (* P3_USABILE *)
  ANDN %Q0.2              (* P3_CMD *)
  S %Q0.2                 (* P3_CMD *)
  [ %MW1 := %MW1 + 1 ]    (* NUM_POMPE_COMANDATE, NUM_POMPE_COMANDATE *)
  S %M13                  (* TERZA_POMPA_COMANDATA *)
  // as ST:
  //   _t1 := NUM_POMPE_COMANDATE < NUM_POMPE_DA_COMANDARE AND NUM_POMPE_DA_COMANDARE >= 3 AND (ORDINE_TERZA_POMPA = 3 OR ORDINE_TERZA_POMPA = 0) AND P3_USABILE AND NOT P3_CMD;
  //   IF _t1 THEN P3_CMD := TRUE; END_IF;
  //   IF _t1 THEN NUM_POMPE_COMANDATE := NUM_POMPE_COMANDATE + 1; END_IF;
  //   IF _t1 THEN TERZA_POMPA_COMANDATA := TRUE; END_IF;

// Rung 172
// Comanda: Terza Pompa (Pompa 4)
  LD [ %MW1 < %MW0 ]      (* NUM_POMPE_COMANDATE, NUM_POMPE_DA_COMANDARE *)
  AND [ %MW0 >= 3 ]       (* NUM_POMPE_DA_COMANDARE *)
  AND( [ %MW10 = 4 ]      (* ORDINE_TERZA_POMPA *)
  OR [ %MW10 = 0 ]        (* ORDINE_TERZA_POMPA *)
  )
  AND %M5                 (* P4_USABILE *)
  ANDN %Q0.3              (* P4_CMD *)
  S %Q0.3                 (* P4_CMD *)
  [ %MW1 := %MW1 + 1 ]    (* NUM_POMPE_COMANDATE, NUM_POMPE_COMANDATE *)
  S %M13                  (* TERZA_POMPA_COMANDATA *)
  // as ST:
  //   _t1 := NUM_POMPE_COMANDATE < NUM_POMPE_DA_COMANDARE AND NUM_POMPE_DA_COMANDARE >= 3 AND (ORDINE_TERZA_POMPA = 4 OR ORDINE_TERZA_POMPA = 0) AND P4_USABILE AND NOT P4_CMD;
  //   IF _t1 THEN P4_CMD := TRUE; END_IF;
  //   IF _t1 THEN NUM_POMPE_COMANDATE := NUM_POMPE_COMANDATE + 1; END_IF;
  //   IF _t1 THEN TERZA_POMPA_COMANDATA := TRUE; END_IF;

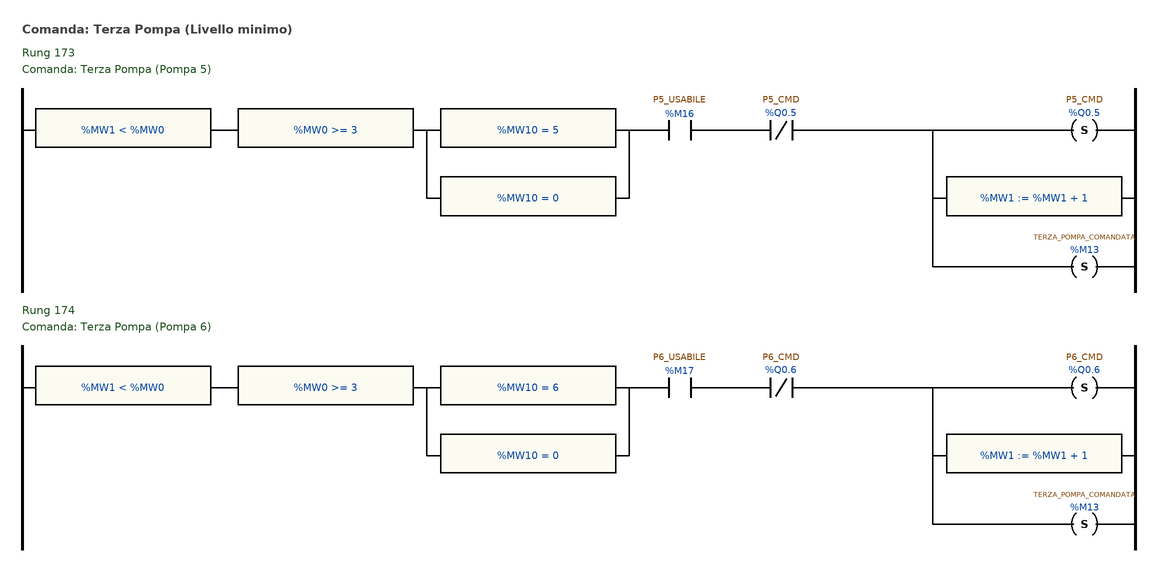

// Rung 173
// Comanda: Terza Pompa (Pompa 5)
  LD [ %MW1 < %MW0 ]      (* NUM_POMPE_COMANDATE, NUM_POMPE_DA_COMANDARE *)
  AND [ %MW0 >= 3 ]       (* NUM_POMPE_DA_COMANDARE *)
  AND( [ %MW10 = 5 ]      (* ORDINE_TERZA_POMPA *)
  OR [ %MW10 = 0 ]        (* ORDINE_TERZA_POMPA *)
  )
  AND %M16                (* P5_USABILE *)
  ANDN %Q0.5              (* P5_CMD *)
  S %Q0.5                 (* P5_CMD *)
  [ %MW1 := %MW1 + 1 ]    (* NUM_POMPE_COMANDATE, NUM_POMPE_COMANDATE *)
  S %M13                  (* TERZA_POMPA_COMANDATA *)
  // as ST:
  //   _t1 := NUM_POMPE_COMANDATE < NUM_POMPE_DA_COMANDARE AND NUM_POMPE_DA_COMANDARE >= 3 AND (ORDINE_TERZA_POMPA = 5 OR ORDINE_TERZA_POMPA = 0) AND P5_USABILE AND NOT P5_CMD;
  //   IF _t1 THEN P5_CMD := TRUE; END_IF;
  //   IF _t1 THEN NUM_POMPE_COMANDATE := NUM_POMPE_COMANDATE + 1; END_IF;
  //   IF _t1 THEN TERZA_POMPA_COMANDATA := TRUE; END_IF;

// Rung 174
// Comanda: Terza Pompa (Pompa 6)
  LD [ %MW1 < %MW0 ]      (* NUM_POMPE_COMANDATE, NUM_POMPE_DA_COMANDARE *)
  AND [ %MW0 >= 3 ]       (* NUM_POMPE_DA_COMANDARE *)
  AND( [ %MW10 = 6 ]      (* ORDINE_TERZA_POMPA *)
  OR [ %MW10 = 0 ]        (* ORDINE_TERZA_POMPA *)
  )
  AND %M17                (* P6_USABILE *)
  ANDN %Q0.6              (* P6_CMD *)
  S %Q0.6                 (* P6_CMD *)
  [ %MW1 := %MW1 + 1 ]    (* NUM_POMPE_COMANDATE, NUM_POMPE_COMANDATE *)
  S %M13                  (* TERZA_POMPA_COMANDATA *)
  // as ST:
  //   _t1 := NUM_POMPE_COMANDATE < NUM_POMPE_DA_COMANDARE AND NUM_POMPE_DA_COMANDARE >= 3 AND (ORDINE_TERZA_POMPA = 6 OR ORDINE_TERZA_POMPA = 0) AND P6_USABILE AND NOT P6_CMD;
  //   IF _t1 THEN P6_CMD := TRUE; END_IF;
  //   IF _t1 THEN NUM_POMPE_COMANDATE := NUM_POMPE_COMANDATE + 1; END_IF;
  //   IF _t1 THEN TERZA_POMPA_COMANDATA := TRUE; END_IF;

Subroutine Ordine: Quarta Pompa (Livello minimo)
  (* SectionNumber=24, Number=22 *)

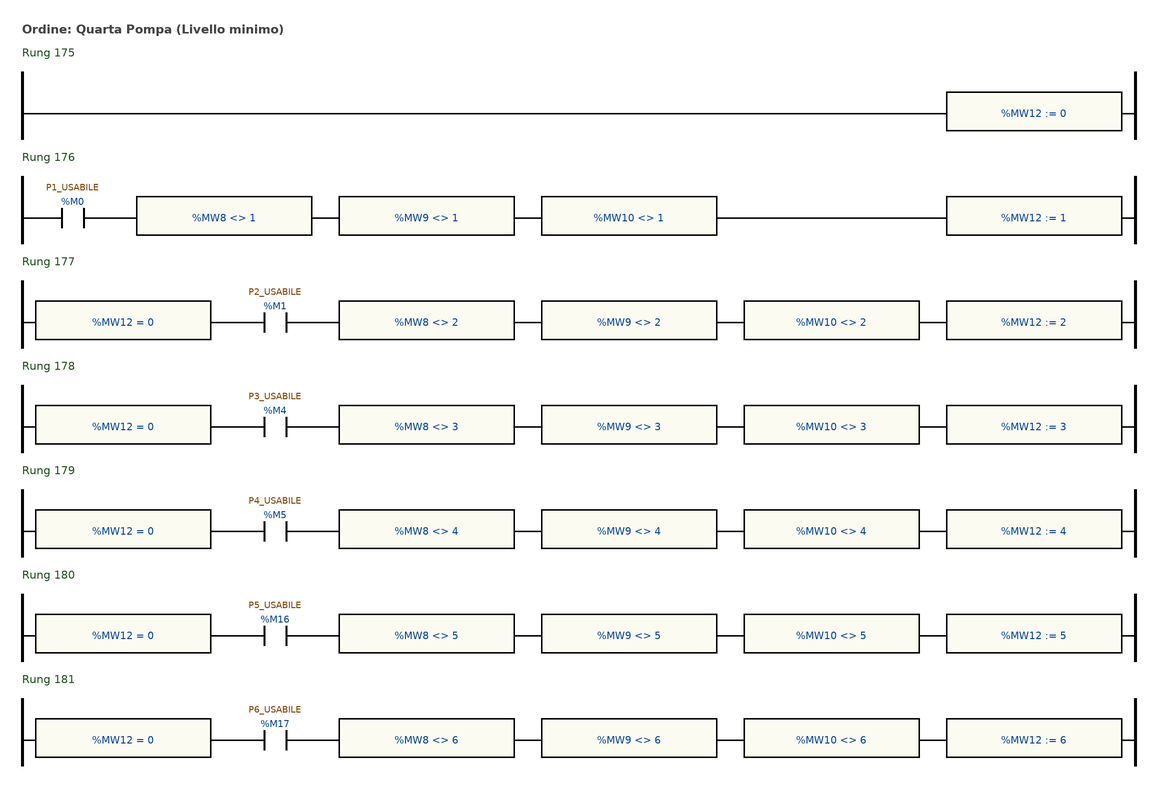

// Rung 175
  LD 1
  [ %MW12 := 0 ]          (* ORDINE_QUARTA_POMPA *)
  // as ST:
  //   ORDINE_QUARTA_POMPA := 0;

// Rung 176
  LD %M0                  (* P1_USABILE *)
  AND [ %MW8 <> 1 ]       (* ORDINE_PRIMA_POMPA *)
  AND [ %MW9 <> 1 ]       (* ORDINE_SECONDA_POMPA *)
  AND [ %MW10 <> 1 ]      (* ORDINE_TERZA_POMPA *)
  [ %MW12 := 1 ]          (* ORDINE_QUARTA_POMPA *)
  // as ST:
  //   IF P1_USABILE AND ORDINE_PRIMA_POMPA <> 1 AND ORDINE_SECONDA_POMPA <> 1 AND ORDINE_TERZA_POMPA <> 1 THEN ORDINE_QUARTA_POMPA := 1; END_IF;

// Rung 177
  LD [ %MW12 = 0 ]        (* ORDINE_QUARTA_POMPA *)
  AND %M1                 (* P2_USABILE *)
  AND [ %MW8 <> 2 ]       (* ORDINE_PRIMA_POMPA *)
  AND [ %MW9 <> 2 ]       (* ORDINE_SECONDA_POMPA *)
  AND [ %MW10 <> 2 ]      (* ORDINE_TERZA_POMPA *)
  [ %MW12 := 2 ]          (* ORDINE_QUARTA_POMPA *)
  // as ST:
  //   IF ORDINE_QUARTA_POMPA = 0 AND P2_USABILE AND ORDINE_PRIMA_POMPA <> 2 AND ORDINE_SECONDA_POMPA <> 2 AND ORDINE_TERZA_POMPA <> 2 THEN ORDINE_QUARTA_POMPA := 2; END_IF;

// Rung 178
  LD [ %MW12 = 0 ]        (* ORDINE_QUARTA_POMPA *)
  AND %M4                 (* P3_USABILE *)
  AND [ %MW8 <> 3 ]       (* ORDINE_PRIMA_POMPA *)
  AND [ %MW9 <> 3 ]       (* ORDINE_SECONDA_POMPA *)
  AND [ %MW10 <> 3 ]      (* ORDINE_TERZA_POMPA *)
  [ %MW12 := 3 ]          (* ORDINE_QUARTA_POMPA *)
  // as ST:
  //   IF ORDINE_QUARTA_POMPA = 0 AND P3_USABILE AND ORDINE_PRIMA_POMPA <> 3 AND ORDINE_SECONDA_POMPA <> 3 AND ORDINE_TERZA_POMPA <> 3 THEN ORDINE_QUARTA_POMPA := 3; END_IF;

// Rung 179
  LD [ %MW12 = 0 ]        (* ORDINE_QUARTA_POMPA *)
  AND %M5                 (* P4_USABILE *)
  AND [ %MW8 <> 4 ]       (* ORDINE_PRIMA_POMPA *)
  AND [ %MW9 <> 4 ]       (* ORDINE_SECONDA_POMPA *)
  AND [ %MW10 <> 4 ]      (* ORDINE_TERZA_POMPA *)
  [ %MW12 := 4 ]          (* ORDINE_QUARTA_POMPA *)
  // as ST:
  //   IF ORDINE_QUARTA_POMPA = 0 AND P4_USABILE AND ORDINE_PRIMA_POMPA <> 4 AND ORDINE_SECONDA_POMPA <> 4 AND ORDINE_TERZA_POMPA <> 4 THEN ORDINE_QUARTA_POMPA := 4; END_IF;

// Rung 180
  LD [ %MW12 = 0 ]        (* ORDINE_QUARTA_POMPA *)
  AND %M16                (* P5_USABILE *)
  AND [ %MW8 <> 5 ]       (* ORDINE_PRIMA_POMPA *)
  AND [ %MW9 <> 5 ]       (* ORDINE_SECONDA_POMPA *)
  AND [ %MW10 <> 5 ]      (* ORDINE_TERZA_POMPA *)
  [ %MW12 := 5 ]          (* ORDINE_QUARTA_POMPA *)
  // as ST:
  //   IF ORDINE_QUARTA_POMPA = 0 AND P5_USABILE AND ORDINE_PRIMA_POMPA <> 5 AND ORDINE_SECONDA_POMPA <> 5 AND ORDINE_TERZA_POMPA <> 5 THEN ORDINE_QUARTA_POMPA := 5; END_IF;

// Rung 181
  LD [ %MW12 = 0 ]        (* ORDINE_QUARTA_POMPA *)
  AND %M17                (* P6_USABILE *)
  AND [ %MW8 <> 6 ]       (* ORDINE_PRIMA_POMPA *)
  AND [ %MW9 <> 6 ]       (* ORDINE_SECONDA_POMPA *)
  AND [ %MW10 <> 6 ]      (* ORDINE_TERZA_POMPA *)
  [ %MW12 := 6 ]          (* ORDINE_QUARTA_POMPA *)
  // as ST:
  //   IF ORDINE_QUARTA_POMPA = 0 AND P6_USABILE AND ORDINE_PRIMA_POMPA <> 6 AND ORDINE_SECONDA_POMPA <> 6 AND ORDINE_TERZA_POMPA <> 6 THEN ORDINE_QUARTA_POMPA := 6; END_IF;

Subroutine Ordine: Quinta Pompa (Livello minimo)
  (* SectionNumber=25, Number=23 *)

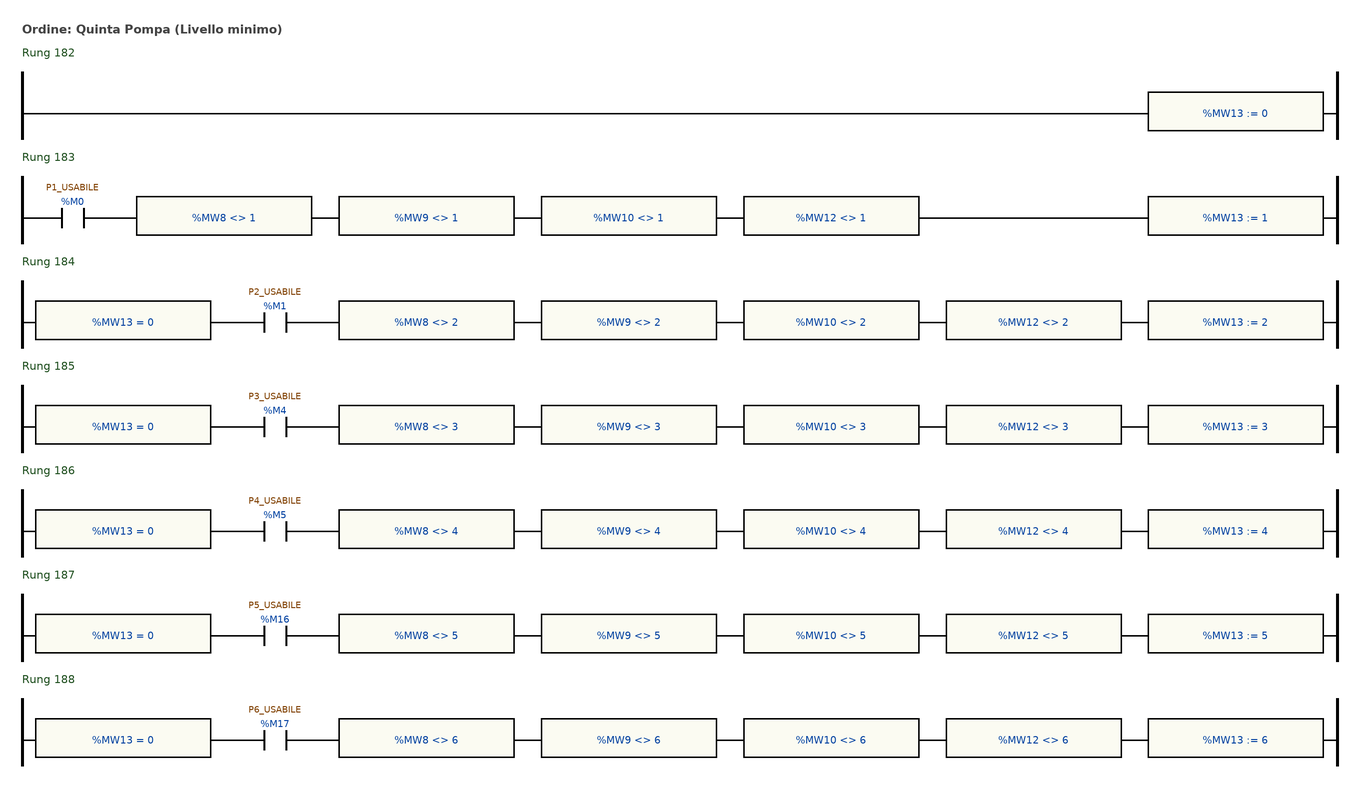

// Rung 182
  LD 1
  [ %MW13 := 0 ]          (* ORDINE_QUINTA_POMPA *)
  // as ST:
  //   ORDINE_QUINTA_POMPA := 0;

// Rung 183
  LD %M0                  (* P1_USABILE *)
  AND [ %MW8 <> 1 ]       (* ORDINE_PRIMA_POMPA *)
  AND [ %MW9 <> 1 ]       (* ORDINE_SECONDA_POMPA *)
  AND [ %MW10 <> 1 ]      (* ORDINE_TERZA_POMPA *)
  AND [ %MW12 <> 1 ]      (* ORDINE_QUARTA_POMPA *)
  [ %MW13 := 1 ]          (* ORDINE_QUINTA_POMPA *)
  // as ST:
  //   IF P1_USABILE AND ORDINE_PRIMA_POMPA <> 1 AND ORDINE_SECONDA_POMPA <> 1 AND ORDINE_TERZA_POMPA <> 1 AND ORDINE_QUARTA_POMPA <> 1 THEN ORDINE_QUINTA_POMPA := 1; END_IF;

// Rung 184
  LD [ %MW13 = 0 ]        (* ORDINE_QUINTA_POMPA *)
  AND %M1                 (* P2_USABILE *)
  AND [ %MW8 <> 2 ]       (* ORDINE_PRIMA_POMPA *)
  AND [ %MW9 <> 2 ]       (* ORDINE_SECONDA_POMPA *)
  AND [ %MW10 <> 2 ]      (* ORDINE_TERZA_POMPA *)
  AND [ %MW12 <> 2 ]      (* ORDINE_QUARTA_POMPA *)
  [ %MW13 := 2 ]          (* ORDINE_QUINTA_POMPA *)
  // as ST:
  //   IF ORDINE_QUINTA_POMPA = 0 AND P2_USABILE AND ORDINE_PRIMA_POMPA <> 2 AND ORDINE_SECONDA_POMPA <> 2 AND ORDINE_TERZA_POMPA <> 2 AND ORDINE_QUARTA_POMPA <> 2 THEN ORDINE_QUINTA_POMPA := 2; END_IF;

// Rung 185
  LD [ %MW13 = 0 ]        (* ORDINE_QUINTA_POMPA *)
  AND %M4                 (* P3_USABILE *)
  AND [ %MW8 <> 3 ]       (* ORDINE_PRIMA_POMPA *)
  AND [ %MW9 <> 3 ]       (* ORDINE_SECONDA_POMPA *)
  AND [ %MW10 <> 3 ]      (* ORDINE_TERZA_POMPA *)
  AND [ %MW12 <> 3 ]      (* ORDINE_QUARTA_POMPA *)
  [ %MW13 := 3 ]          (* ORDINE_QUINTA_POMPA *)
  // as ST:
  //   IF ORDINE_QUINTA_POMPA = 0 AND P3_USABILE AND ORDINE_PRIMA_POMPA <> 3 AND ORDINE_SECONDA_POMPA <> 3 AND ORDINE_TERZA_POMPA <> 3 AND ORDINE_QUARTA_POMPA <> 3 THEN ORDINE_QUINTA_POMPA := 3; END_IF;

// Rung 186
  LD [ %MW13 = 0 ]        (* ORDINE_QUINTA_POMPA *)
  AND %M5                 (* P4_USABILE *)
  AND [ %MW8 <> 4 ]       (* ORDINE_PRIMA_POMPA *)
  AND [ %MW9 <> 4 ]       (* ORDINE_SECONDA_POMPA *)
  AND [ %MW10 <> 4 ]      (* ORDINE_TERZA_POMPA *)
  AND [ %MW12 <> 4 ]      (* ORDINE_QUARTA_POMPA *)
  [ %MW13 := 4 ]          (* ORDINE_QUINTA_POMPA *)
  // as ST:
  //   IF ORDINE_QUINTA_POMPA = 0 AND P4_USABILE AND ORDINE_PRIMA_POMPA <> 4 AND ORDINE_SECONDA_POMPA <> 4 AND ORDINE_TERZA_POMPA <> 4 AND ORDINE_QUARTA_POMPA <> 4 THEN ORDINE_QUINTA_POMPA := 4; END_IF;

// Rung 187
  LD [ %MW13 = 0 ]        (* ORDINE_QUINTA_POMPA *)
  AND %M16                (* P5_USABILE *)
  AND [ %MW8 <> 5 ]       (* ORDINE_PRIMA_POMPA *)
  AND [ %MW9 <> 5 ]       (* ORDINE_SECONDA_POMPA *)
  AND [ %MW10 <> 5 ]      (* ORDINE_TERZA_POMPA *)
  AND [ %MW12 <> 5 ]      (* ORDINE_QUARTA_POMPA *)
  [ %MW13 := 5 ]          (* ORDINE_QUINTA_POMPA *)
  // as ST:
  //   IF ORDINE_QUINTA_POMPA = 0 AND P5_USABILE AND ORDINE_PRIMA_POMPA <> 5 AND ORDINE_SECONDA_POMPA <> 5 AND ORDINE_TERZA_POMPA <> 5 AND ORDINE_QUARTA_POMPA <> 5 THEN ORDINE_QUINTA_POMPA := 5; END_IF;

// Rung 188
  LD [ %MW13 = 0 ]        (* ORDINE_QUINTA_POMPA *)
  AND %M17                (* P6_USABILE *)
  AND [ %MW8 <> 6 ]       (* ORDINE_PRIMA_POMPA *)
  AND [ %MW9 <> 6 ]       (* ORDINE_SECONDA_POMPA *)
  AND [ %MW10 <> 6 ]      (* ORDINE_TERZA_POMPA *)
  AND [ %MW12 <> 6 ]      (* ORDINE_QUARTA_POMPA *)
  [ %MW13 := 6 ]          (* ORDINE_QUINTA_POMPA *)
  // as ST:
  //   IF ORDINE_QUINTA_POMPA = 0 AND P6_USABILE AND ORDINE_PRIMA_POMPA <> 6 AND ORDINE_SECONDA_POMPA <> 6 AND ORDINE_TERZA_POMPA <> 6 AND ORDINE_QUARTA_POMPA <> 6 THEN ORDINE_QUINTA_POMPA := 6; END_IF;

Subroutine Comanda: Quarta Pompa (Livello minimo)
  (* SectionNumber=26, Number=24 *)

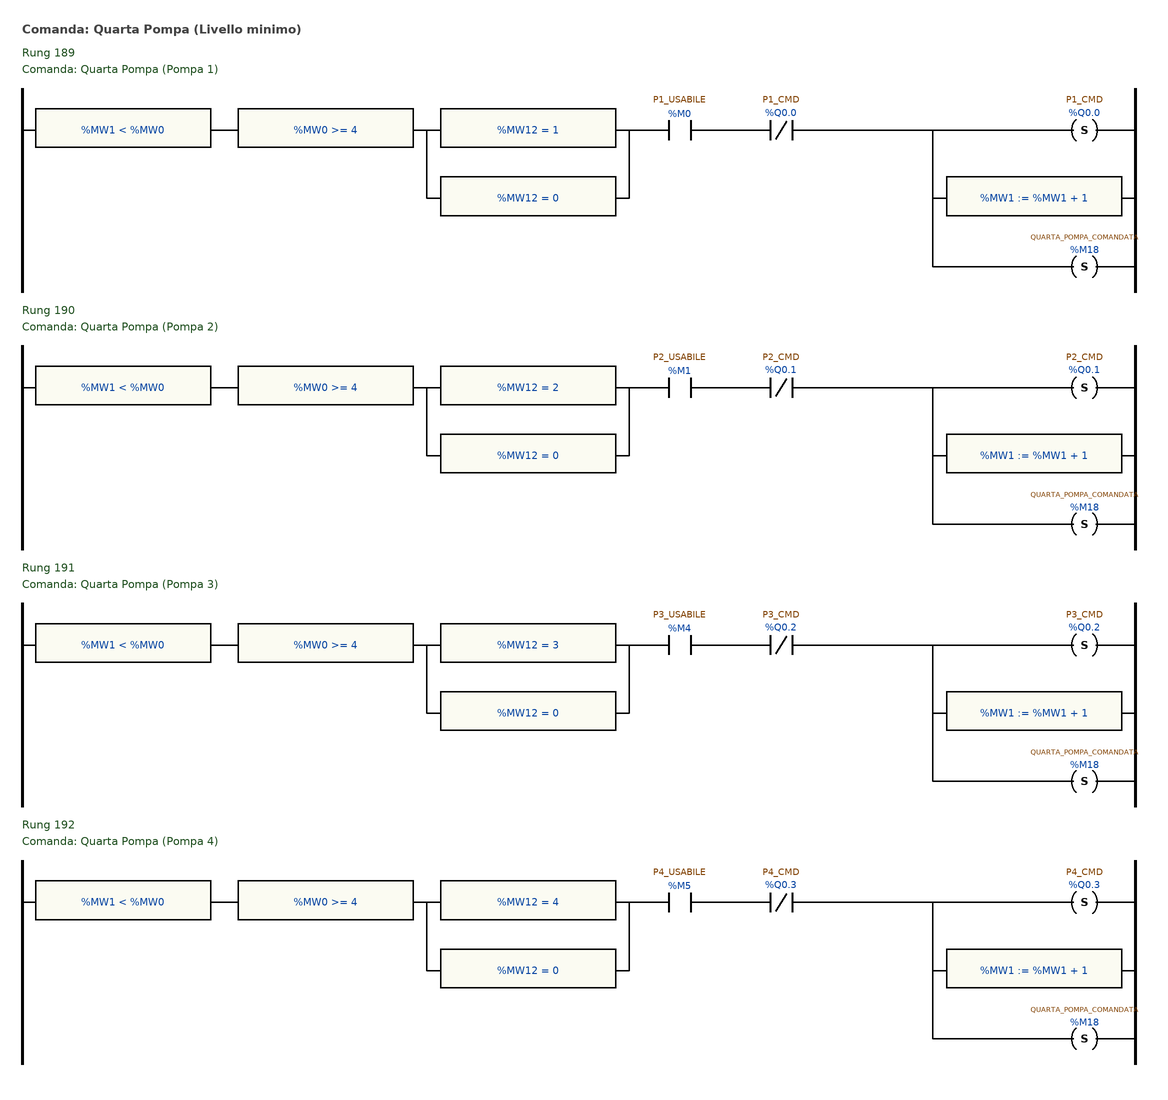

// Rung 189
// Comanda: Quarta Pompa (Pompa 1)
  LD [ %MW1 < %MW0 ]      (* NUM_POMPE_COMANDATE, NUM_POMPE_DA_COMANDARE *)
  AND [ %MW0 >= 4 ]       (* NUM_POMPE_DA_COMANDARE *)
  AND( [ %MW12 = 1 ]      (* ORDINE_QUARTA_POMPA *)
  OR [ %MW12 = 0 ]        (* ORDINE_QUARTA_POMPA *)
  )
  AND %M0                 (* P1_USABILE *)
  ANDN %Q0.0              (* P1_CMD *)
  S %Q0.0                 (* P1_CMD *)
  [ %MW1 := %MW1 + 1 ]    (* NUM_POMPE_COMANDATE, NUM_POMPE_COMANDATE *)
  S %M18                  (* QUARTA_POMPA_COMANDATA *)
  // as ST:
  //   _t1 := NUM_POMPE_COMANDATE < NUM_POMPE_DA_COMANDARE AND NUM_POMPE_DA_COMANDARE >= 4 AND (ORDINE_QUARTA_POMPA = 1 OR ORDINE_QUARTA_POMPA = 0) AND P1_USABILE AND NOT P1_CMD;
  //   IF _t1 THEN P1_CMD := TRUE; END_IF;
  //   IF _t1 THEN NUM_POMPE_COMANDATE := NUM_POMPE_COMANDATE + 1; END_IF;
  //   IF _t1 THEN QUARTA_POMPA_COMANDATA := TRUE; END_IF;

// Rung 190
// Comanda: Quarta Pompa (Pompa 2)
  LD [ %MW1 < %MW0 ]      (* NUM_POMPE_COMANDATE, NUM_POMPE_DA_COMANDARE *)
  AND [ %MW0 >= 4 ]       (* NUM_POMPE_DA_COMANDARE *)
  AND( [ %MW12 = 2 ]      (* ORDINE_QUARTA_POMPA *)
  OR [ %MW12 = 0 ]        (* ORDINE_QUARTA_POMPA *)
  )
  AND %M1                 (* P2_USABILE *)
  ANDN %Q0.1              (* P2_CMD *)
  S %Q0.1                 (* P2_CMD *)
  [ %MW1 := %MW1 + 1 ]    (* NUM_POMPE_COMANDATE, NUM_POMPE_COMANDATE *)
  S %M18                  (* QUARTA_POMPA_COMANDATA *)
  // as ST:
  //   _t1 := NUM_POMPE_COMANDATE < NUM_POMPE_DA_COMANDARE AND NUM_POMPE_DA_COMANDARE >= 4 AND (ORDINE_QUARTA_POMPA = 2 OR ORDINE_QUARTA_POMPA = 0) AND P2_USABILE AND NOT P2_CMD;
  //   IF _t1 THEN P2_CMD := TRUE; END_IF;
  //   IF _t1 THEN NUM_POMPE_COMANDATE := NUM_POMPE_COMANDATE + 1; END_IF;
  //   IF _t1 THEN QUARTA_POMPA_COMANDATA := TRUE; END_IF;

// Rung 191
// Comanda: Quarta Pompa (Pompa 3)
  LD [ %MW1 < %MW0 ]      (* NUM_POMPE_COMANDATE, NUM_POMPE_DA_COMANDARE *)
  AND [ %MW0 >= 4 ]       (* NUM_POMPE_DA_COMANDARE *)
  AND( [ %MW12 = 3 ]      (* ORDINE_QUARTA_POMPA *)
  OR [ %MW12 = 0 ]        (* ORDINE_QUARTA_POMPA *)
  )
  AND %M4                 (* P3_USABILE *)
  ANDN %Q0.2              (* P3_CMD *)
  S %Q0.2                 (* P3_CMD *)
  [ %MW1 := %MW1 + 1 ]    (* NUM_POMPE_COMANDATE, NUM_POMPE_COMANDATE *)
  S %M18                  (* QUARTA_POMPA_COMANDATA *)
  // as ST:
  //   _t1 := NUM_POMPE_COMANDATE < NUM_POMPE_DA_COMANDARE AND NUM_POMPE_DA_COMANDARE >= 4 AND (ORDINE_QUARTA_POMPA = 3 OR ORDINE_QUARTA_POMPA = 0) AND P3_USABILE AND NOT P3_CMD;
  //   IF _t1 THEN P3_CMD := TRUE; END_IF;
  //   IF _t1 THEN NUM_POMPE_COMANDATE := NUM_POMPE_COMANDATE + 1; END_IF;
  //   IF _t1 THEN QUARTA_POMPA_COMANDATA := TRUE; END_IF;

// Rung 192
// Comanda: Quarta Pompa (Pompa 4)
  LD [ %MW1 < %MW0 ]      (* NUM_POMPE_COMANDATE, NUM_POMPE_DA_COMANDARE *)
  AND [ %MW0 >= 4 ]       (* NUM_POMPE_DA_COMANDARE *)
  AND( [ %MW12 = 4 ]      (* ORDINE_QUARTA_POMPA *)
  OR [ %MW12 = 0 ]        (* ORDINE_QUARTA_POMPA *)
  )
  AND %M5                 (* P4_USABILE *)
  ANDN %Q0.3              (* P4_CMD *)
  S %Q0.3                 (* P4_CMD *)
  [ %MW1 := %MW1 + 1 ]    (* NUM_POMPE_COMANDATE, NUM_POMPE_COMANDATE *)
  S %M18                  (* QUARTA_POMPA_COMANDATA *)
  // as ST:
  //   _t1 := NUM_POMPE_COMANDATE < NUM_POMPE_DA_COMANDARE AND NUM_POMPE_DA_COMANDARE >= 4 AND (ORDINE_QUARTA_POMPA = 4 OR ORDINE_QUARTA_POMPA = 0) AND P4_USABILE AND NOT P4_CMD;
  //   IF _t1 THEN P4_CMD := TRUE; END_IF;
  //   IF _t1 THEN NUM_POMPE_COMANDATE := NUM_POMPE_COMANDATE + 1; END_IF;
  //   IF _t1 THEN QUARTA_POMPA_COMANDATA := TRUE; END_IF;

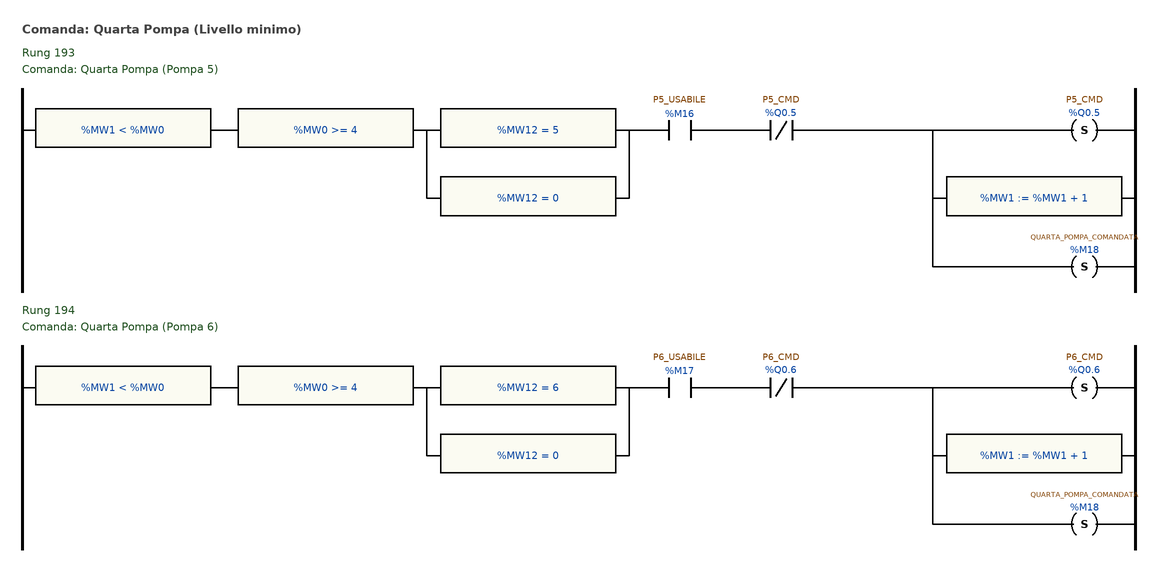

// Rung 193
// Comanda: Quarta Pompa (Pompa 5)
  LD [ %MW1 < %MW0 ]      (* NUM_POMPE_COMANDATE, NUM_POMPE_DA_COMANDARE *)
  AND [ %MW0 >= 4 ]       (* NUM_POMPE_DA_COMANDARE *)
  AND( [ %MW12 = 5 ]      (* ORDINE_QUARTA_POMPA *)
  OR [ %MW12 = 0 ]        (* ORDINE_QUARTA_POMPA *)
  )
  AND %M16                (* P5_USABILE *)
  ANDN %Q0.5              (* P5_CMD *)
  S %Q0.5                 (* P5_CMD *)
  [ %MW1 := %MW1 + 1 ]    (* NUM_POMPE_COMANDATE, NUM_POMPE_COMANDATE *)
  S %M18                  (* QUARTA_POMPA_COMANDATA *)
  // as ST:
  //   _t1 := NUM_POMPE_COMANDATE < NUM_POMPE_DA_COMANDARE AND NUM_POMPE_DA_COMANDARE >= 4 AND (ORDINE_QUARTA_POMPA = 5 OR ORDINE_QUARTA_POMPA = 0) AND P5_USABILE AND NOT P5_CMD;
  //   IF _t1 THEN P5_CMD := TRUE; END_IF;
  //   IF _t1 THEN NUM_POMPE_COMANDATE := NUM_POMPE_COMANDATE + 1; END_IF;
  //   IF _t1 THEN QUARTA_POMPA_COMANDATA := TRUE; END_IF;

// Rung 194
// Comanda: Quarta Pompa (Pompa 6)
  LD [ %MW1 < %MW0 ]      (* NUM_POMPE_COMANDATE, NUM_POMPE_DA_COMANDARE *)
  AND [ %MW0 >= 4 ]       (* NUM_POMPE_DA_COMANDARE *)
  AND( [ %MW12 = 6 ]      (* ORDINE_QUARTA_POMPA *)
  OR [ %MW12 = 0 ]        (* ORDINE_QUARTA_POMPA *)
  )
  AND %M17                (* P6_USABILE *)
  ANDN %Q0.6              (* P6_CMD *)
  S %Q0.6                 (* P6_CMD *)
  [ %MW1 := %MW1 + 1 ]    (* NUM_POMPE_COMANDATE, NUM_POMPE_COMANDATE *)
  S %M18                  (* QUARTA_POMPA_COMANDATA *)
  // as ST:
  //   _t1 := NUM_POMPE_COMANDATE < NUM_POMPE_DA_COMANDARE AND NUM_POMPE_DA_COMANDARE >= 4 AND (ORDINE_QUARTA_POMPA = 6 OR ORDINE_QUARTA_POMPA = 0) AND P6_USABILE AND NOT P6_CMD;
  //   IF _t1 THEN P6_CMD := TRUE; END_IF;
  //   IF _t1 THEN NUM_POMPE_COMANDATE := NUM_POMPE_COMANDATE + 1; END_IF;
  //   IF _t1 THEN QUARTA_POMPA_COMANDATA := TRUE; END_IF;

Subroutine Comanda: Quinta Pompa (Livello minimo)
  (* SectionNumber=27, Number=25 *)

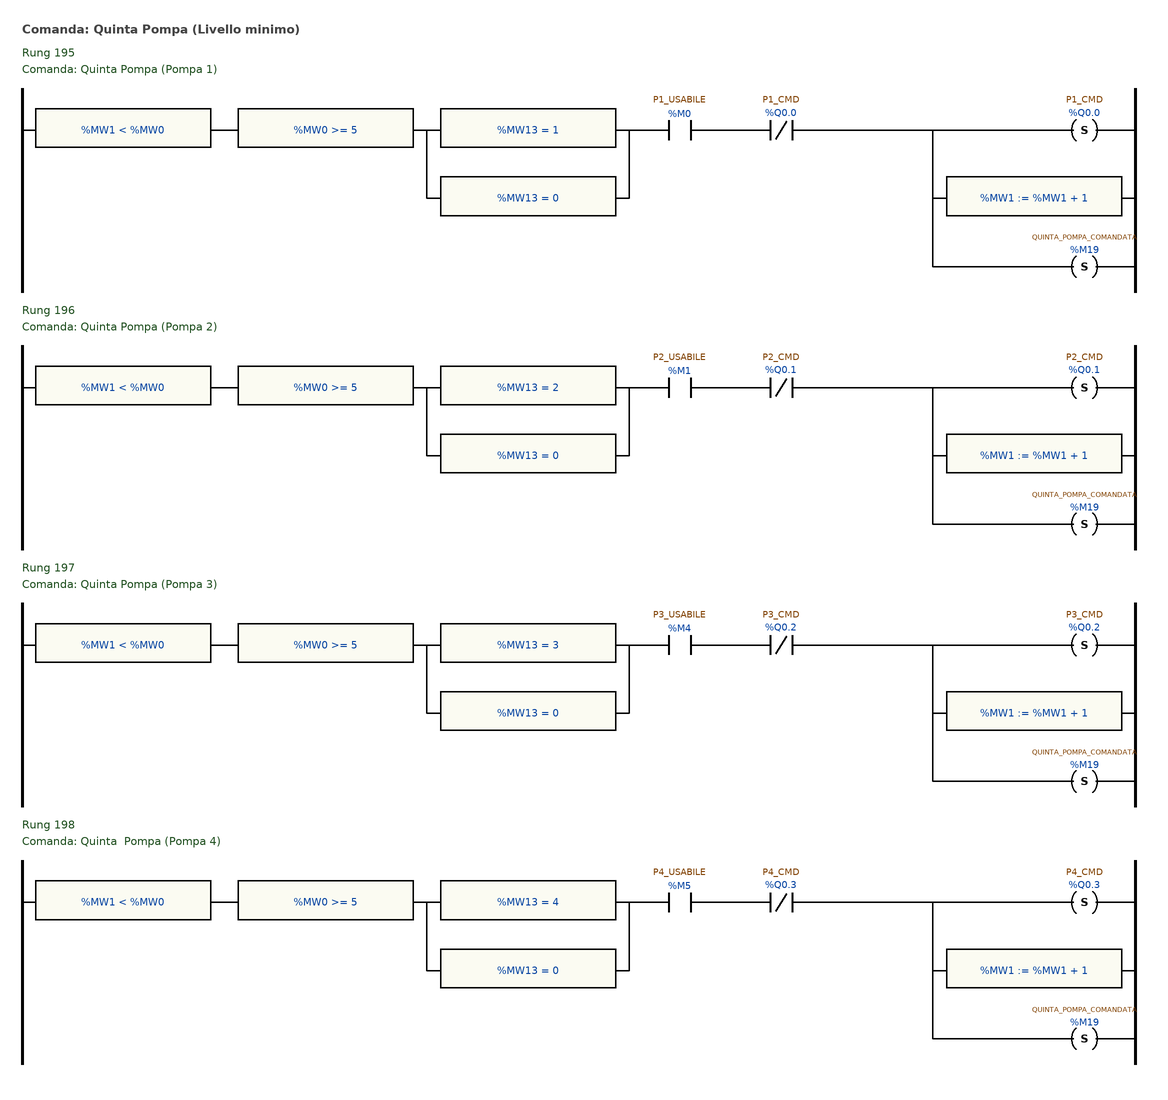

// Rung 195
// Comanda: Quinta Pompa (Pompa 1)
  LD [ %MW1 < %MW0 ]      (* NUM_POMPE_COMANDATE, NUM_POMPE_DA_COMANDARE *)
  AND [ %MW0 >= 5 ]       (* NUM_POMPE_DA_COMANDARE *)
  AND( [ %MW13 = 1 ]      (* ORDINE_QUINTA_POMPA *)
  OR [ %MW13 = 0 ]        (* ORDINE_QUINTA_POMPA *)
  )
  AND %M0                 (* P1_USABILE *)
  ANDN %Q0.0              (* P1_CMD *)
  S %Q0.0                 (* P1_CMD *)
  [ %MW1 := %MW1 + 1 ]    (* NUM_POMPE_COMANDATE, NUM_POMPE_COMANDATE *)
  S %M19                  (* QUINTA_POMPA_COMANDATA *)
  // as ST:
  //   _t1 := NUM_POMPE_COMANDATE < NUM_POMPE_DA_COMANDARE AND NUM_POMPE_DA_COMANDARE >= 5 AND (ORDINE_QUINTA_POMPA = 1 OR ORDINE_QUINTA_POMPA = 0) AND P1_USABILE AND NOT P1_CMD;
  //   IF _t1 THEN P1_CMD := TRUE; END_IF;
  //   IF _t1 THEN NUM_POMPE_COMANDATE := NUM_POMPE_COMANDATE + 1; END_IF;
  //   IF _t1 THEN QUINTA_POMPA_COMANDATA := TRUE; END_IF;

// Rung 196
// Comanda: Quinta Pompa (Pompa 2)
  LD [ %MW1 < %MW0 ]      (* NUM_POMPE_COMANDATE, NUM_POMPE_DA_COMANDARE *)
  AND [ %MW0 >= 5 ]       (* NUM_POMPE_DA_COMANDARE *)
  AND( [ %MW13 = 2 ]      (* ORDINE_QUINTA_POMPA *)
  OR [ %MW13 = 0 ]        (* ORDINE_QUINTA_POMPA *)
  )
  AND %M1                 (* P2_USABILE *)
  ANDN %Q0.1              (* P2_CMD *)
  S %Q0.1                 (* P2_CMD *)
  [ %MW1 := %MW1 + 1 ]    (* NUM_POMPE_COMANDATE, NUM_POMPE_COMANDATE *)
  S %M19                  (* QUINTA_POMPA_COMANDATA *)
  // as ST:
  //   _t1 := NUM_POMPE_COMANDATE < NUM_POMPE_DA_COMANDARE AND NUM_POMPE_DA_COMANDARE >= 5 AND (ORDINE_QUINTA_POMPA = 2 OR ORDINE_QUINTA_POMPA = 0) AND P2_USABILE AND NOT P2_CMD;
  //   IF _t1 THEN P2_CMD := TRUE; END_IF;
  //   IF _t1 THEN NUM_POMPE_COMANDATE := NUM_POMPE_COMANDATE + 1; END_IF;
  //   IF _t1 THEN QUINTA_POMPA_COMANDATA := TRUE; END_IF;

// Rung 197
// Comanda: Quinta Pompa (Pompa 3)
  LD [ %MW1 < %MW0 ]      (* NUM_POMPE_COMANDATE, NUM_POMPE_DA_COMANDARE *)
  AND [ %MW0 >= 5 ]       (* NUM_POMPE_DA_COMANDARE *)
  AND( [ %MW13 = 3 ]      (* ORDINE_QUINTA_POMPA *)
  OR [ %MW13 = 0 ]        (* ORDINE_QUINTA_POMPA *)
  )
  AND %M4                 (* P3_USABILE *)
  ANDN %Q0.2              (* P3_CMD *)
  S %Q0.2                 (* P3_CMD *)
  [ %MW1 := %MW1 + 1 ]    (* NUM_POMPE_COMANDATE, NUM_POMPE_COMANDATE *)
  S %M19                  (* QUINTA_POMPA_COMANDATA *)
  // as ST:
  //   _t1 := NUM_POMPE_COMANDATE < NUM_POMPE_DA_COMANDARE AND NUM_POMPE_DA_COMANDARE >= 5 AND (ORDINE_QUINTA_POMPA = 3 OR ORDINE_QUINTA_POMPA = 0) AND P3_USABILE AND NOT P3_CMD;
  //   IF _t1 THEN P3_CMD := TRUE; END_IF;
  //   IF _t1 THEN NUM_POMPE_COMANDATE := NUM_POMPE_COMANDATE + 1; END_IF;
  //   IF _t1 THEN QUINTA_POMPA_COMANDATA := TRUE; END_IF;

// Rung 198
// Comanda: Quinta  Pompa (Pompa 4)
  LD [ %MW1 < %MW0 ]      (* NUM_POMPE_COMANDATE, NUM_POMPE_DA_COMANDARE *)
  AND [ %MW0 >= 5 ]       (* NUM_POMPE_DA_COMANDARE *)
  AND( [ %MW13 = 4 ]      (* ORDINE_QUINTA_POMPA *)
  OR [ %MW13 = 0 ]        (* ORDINE_QUINTA_POMPA *)
  )
  AND %M5                 (* P4_USABILE *)
  ANDN %Q0.3              (* P4_CMD *)
  S %Q0.3                 (* P4_CMD *)
  [ %MW1 := %MW1 + 1 ]    (* NUM_POMPE_COMANDATE, NUM_POMPE_COMANDATE *)
  S %M19                  (* QUINTA_POMPA_COMANDATA *)
  // as ST:
  //   _t1 := NUM_POMPE_COMANDATE < NUM_POMPE_DA_COMANDARE AND NUM_POMPE_DA_COMANDARE >= 5 AND (ORDINE_QUINTA_POMPA = 4 OR ORDINE_QUINTA_POMPA = 0) AND P4_USABILE AND NOT P4_CMD;
  //   IF _t1 THEN P4_CMD := TRUE; END_IF;
  //   IF _t1 THEN NUM_POMPE_COMANDATE := NUM_POMPE_COMANDATE + 1; END_IF;
  //   IF _t1 THEN QUINTA_POMPA_COMANDATA := TRUE; END_IF;

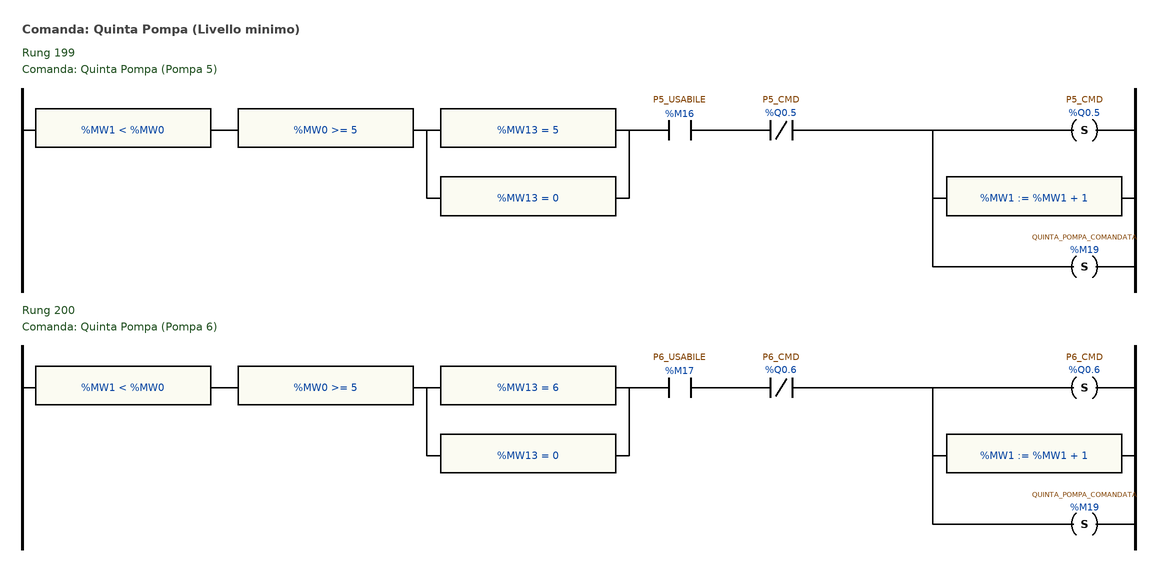

// Rung 199
// Comanda: Quinta Pompa (Pompa 5)
  LD [ %MW1 < %MW0 ]      (* NUM_POMPE_COMANDATE, NUM_POMPE_DA_COMANDARE *)
  AND [ %MW0 >= 5 ]       (* NUM_POMPE_DA_COMANDARE *)
  AND( [ %MW13 = 5 ]      (* ORDINE_QUINTA_POMPA *)
  OR [ %MW13 = 0 ]        (* ORDINE_QUINTA_POMPA *)
  )
  AND %M16                (* P5_USABILE *)
  ANDN %Q0.5              (* P5_CMD *)
  S %Q0.5                 (* P5_CMD *)
  [ %MW1 := %MW1 + 1 ]    (* NUM_POMPE_COMANDATE, NUM_POMPE_COMANDATE *)
  S %M19                  (* QUINTA_POMPA_COMANDATA *)
  // as ST:
  //   _t1 := NUM_POMPE_COMANDATE < NUM_POMPE_DA_COMANDARE AND NUM_POMPE_DA_COMANDARE >= 5 AND (ORDINE_QUINTA_POMPA = 5 OR ORDINE_QUINTA_POMPA = 0) AND P5_USABILE AND NOT P5_CMD;
  //   IF _t1 THEN P5_CMD := TRUE; END_IF;
  //   IF _t1 THEN NUM_POMPE_COMANDATE := NUM_POMPE_COMANDATE + 1; END_IF;
  //   IF _t1 THEN QUINTA_POMPA_COMANDATA := TRUE; END_IF;

// Rung 200
// Comanda: Quinta Pompa (Pompa 6)
  LD [ %MW1 < %MW0 ]      (* NUM_POMPE_COMANDATE, NUM_POMPE_DA_COMANDARE *)
  AND [ %MW0 >= 5 ]       (* NUM_POMPE_DA_COMANDARE *)
  AND( [ %MW13 = 6 ]      (* ORDINE_QUINTA_POMPA *)
  OR [ %MW13 = 0 ]        (* ORDINE_QUINTA_POMPA *)
  )
  AND %M17                (* P6_USABILE *)
  ANDN %Q0.6              (* P6_CMD *)
  S %Q0.6                 (* P6_CMD *)
  [ %MW1 := %MW1 + 1 ]    (* NUM_POMPE_COMANDATE, NUM_POMPE_COMANDATE *)
  S %M19                  (* QUINTA_POMPA_COMANDATA *)
  // as ST:
  //   _t1 := NUM_POMPE_COMANDATE < NUM_POMPE_DA_COMANDARE AND NUM_POMPE_DA_COMANDARE >= 5 AND (ORDINE_QUINTA_POMPA = 6 OR ORDINE_QUINTA_POMPA = 0) AND P6_USABILE AND NOT P6_CMD;
  //   IF _t1 THEN P6_CMD := TRUE; END_IF;
  //   IF _t1 THEN NUM_POMPE_COMANDATE := NUM_POMPE_COMANDATE + 1; END_IF;
  //   IF _t1 THEN QUINTA_POMPA_COMANDATA := TRUE; END_IF;

Subroutine Ordine: Quarta Pompa (Spegnimento graduale)
  (* SectionNumber=28, Number=26 *)

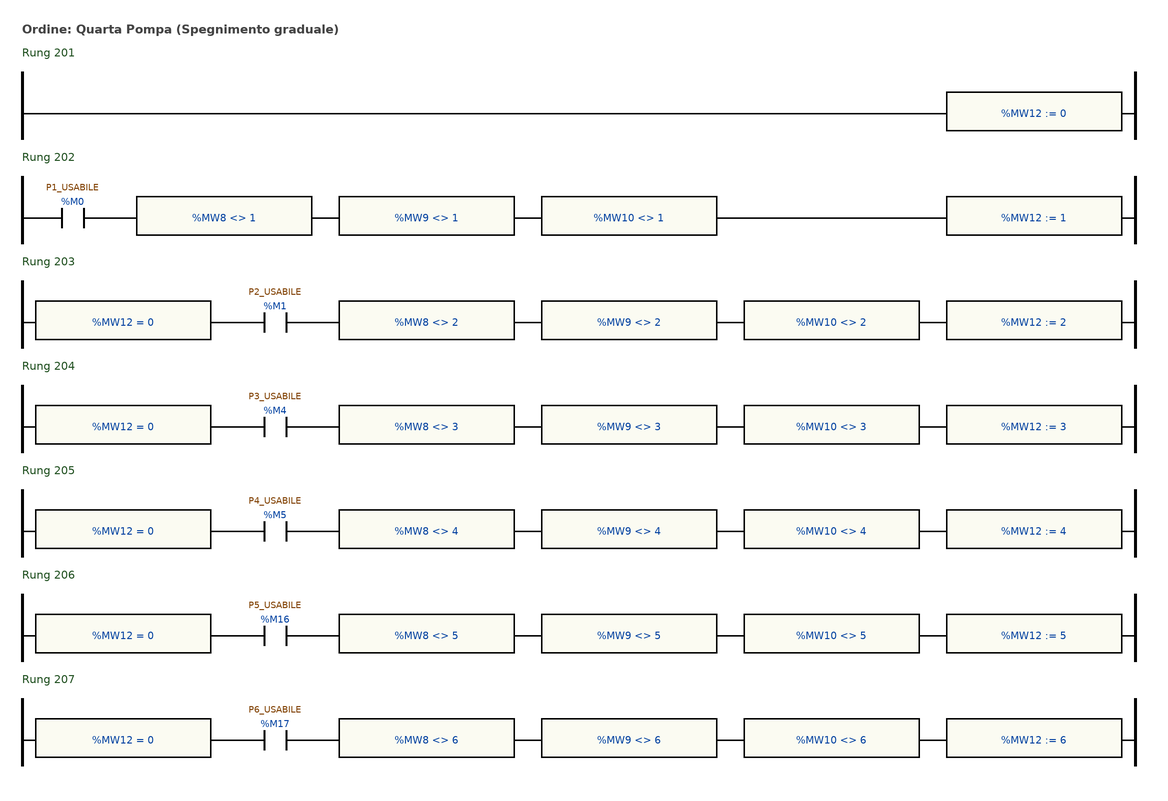

// Rung 201
  LD 1
  [ %MW12 := 0 ]          (* ORDINE_QUARTA_POMPA *)
  // as ST:
  //   ORDINE_QUARTA_POMPA := 0;

// Rung 202
  LD %M0                  (* P1_USABILE *)
  AND [ %MW8 <> 1 ]       (* ORDINE_PRIMA_POMPA *)
  AND [ %MW9 <> 1 ]       (* ORDINE_SECONDA_POMPA *)
  AND [ %MW10 <> 1 ]      (* ORDINE_TERZA_POMPA *)
  [ %MW12 := 1 ]          (* ORDINE_QUARTA_POMPA *)
  // as ST:
  //   IF P1_USABILE AND ORDINE_PRIMA_POMPA <> 1 AND ORDINE_SECONDA_POMPA <> 1 AND ORDINE_TERZA_POMPA <> 1 THEN ORDINE_QUARTA_POMPA := 1; END_IF;

// Rung 203
  LD [ %MW12 = 0 ]        (* ORDINE_QUARTA_POMPA *)
  AND %M1                 (* P2_USABILE *)
  AND [ %MW8 <> 2 ]       (* ORDINE_PRIMA_POMPA *)
  AND [ %MW9 <> 2 ]       (* ORDINE_SECONDA_POMPA *)
  AND [ %MW10 <> 2 ]      (* ORDINE_TERZA_POMPA *)
  [ %MW12 := 2 ]          (* ORDINE_QUARTA_POMPA *)
  // as ST:
  //   IF ORDINE_QUARTA_POMPA = 0 AND P2_USABILE AND ORDINE_PRIMA_POMPA <> 2 AND ORDINE_SECONDA_POMPA <> 2 AND ORDINE_TERZA_POMPA <> 2 THEN ORDINE_QUARTA_POMPA := 2; END_IF;

// Rung 204
  LD [ %MW12 = 0 ]        (* ORDINE_QUARTA_POMPA *)
  AND %M4                 (* P3_USABILE *)
  AND [ %MW8 <> 3 ]       (* ORDINE_PRIMA_POMPA *)
  AND [ %MW9 <> 3 ]       (* ORDINE_SECONDA_POMPA *)
  AND [ %MW10 <> 3 ]      (* ORDINE_TERZA_POMPA *)
  [ %MW12 := 3 ]          (* ORDINE_QUARTA_POMPA *)
  // as ST:
  //   IF ORDINE_QUARTA_POMPA = 0 AND P3_USABILE AND ORDINE_PRIMA_POMPA <> 3 AND ORDINE_SECONDA_POMPA <> 3 AND ORDINE_TERZA_POMPA <> 3 THEN ORDINE_QUARTA_POMPA := 3; END_IF;

// Rung 205
  LD [ %MW12 = 0 ]        (* ORDINE_QUARTA_POMPA *)
  AND %M5                 (* P4_USABILE *)
  AND [ %MW8 <> 4 ]       (* ORDINE_PRIMA_POMPA *)
  AND [ %MW9 <> 4 ]       (* ORDINE_SECONDA_POMPA *)
  AND [ %MW10 <> 4 ]      (* ORDINE_TERZA_POMPA *)
  [ %MW12 := 4 ]          (* ORDINE_QUARTA_POMPA *)
  // as ST:
  //   IF ORDINE_QUARTA_POMPA = 0 AND P4_USABILE AND ORDINE_PRIMA_POMPA <> 4 AND ORDINE_SECONDA_POMPA <> 4 AND ORDINE_TERZA_POMPA <> 4 THEN ORDINE_QUARTA_POMPA := 4; END_IF;

// Rung 206
  LD [ %MW12 = 0 ]        (* ORDINE_QUARTA_POMPA *)
  AND %M16                (* P5_USABILE *)
  AND [ %MW8 <> 5 ]       (* ORDINE_PRIMA_POMPA *)
  AND [ %MW9 <> 5 ]       (* ORDINE_SECONDA_POMPA *)
  AND [ %MW10 <> 5 ]      (* ORDINE_TERZA_POMPA *)
  [ %MW12 := 5 ]          (* ORDINE_QUARTA_POMPA *)
  // as ST:
  //   IF ORDINE_QUARTA_POMPA = 0 AND P5_USABILE AND ORDINE_PRIMA_POMPA <> 5 AND ORDINE_SECONDA_POMPA <> 5 AND ORDINE_TERZA_POMPA <> 5 THEN ORDINE_QUARTA_POMPA := 5; END_IF;

// Rung 207
  LD [ %MW12 = 0 ]        (* ORDINE_QUARTA_POMPA *)
  AND %M17                (* P6_USABILE *)
  AND [ %MW8 <> 6 ]       (* ORDINE_PRIMA_POMPA *)
  AND [ %MW9 <> 6 ]       (* ORDINE_SECONDA_POMPA *)
  AND [ %MW10 <> 6 ]      (* ORDINE_TERZA_POMPA *)
  [ %MW12 := 6 ]          (* ORDINE_QUARTA_POMPA *)
  // as ST:
  //   IF ORDINE_QUARTA_POMPA = 0 AND P6_USABILE AND ORDINE_PRIMA_POMPA <> 6 AND ORDINE_SECONDA_POMPA <> 6 AND ORDINE_TERZA_POMPA <> 6 THEN ORDINE_QUARTA_POMPA := 6; END_IF;

Subroutine Ordine: Quinta Pompa (Spegnimento graduale)
  (* SectionNumber=29, Number=27 *)

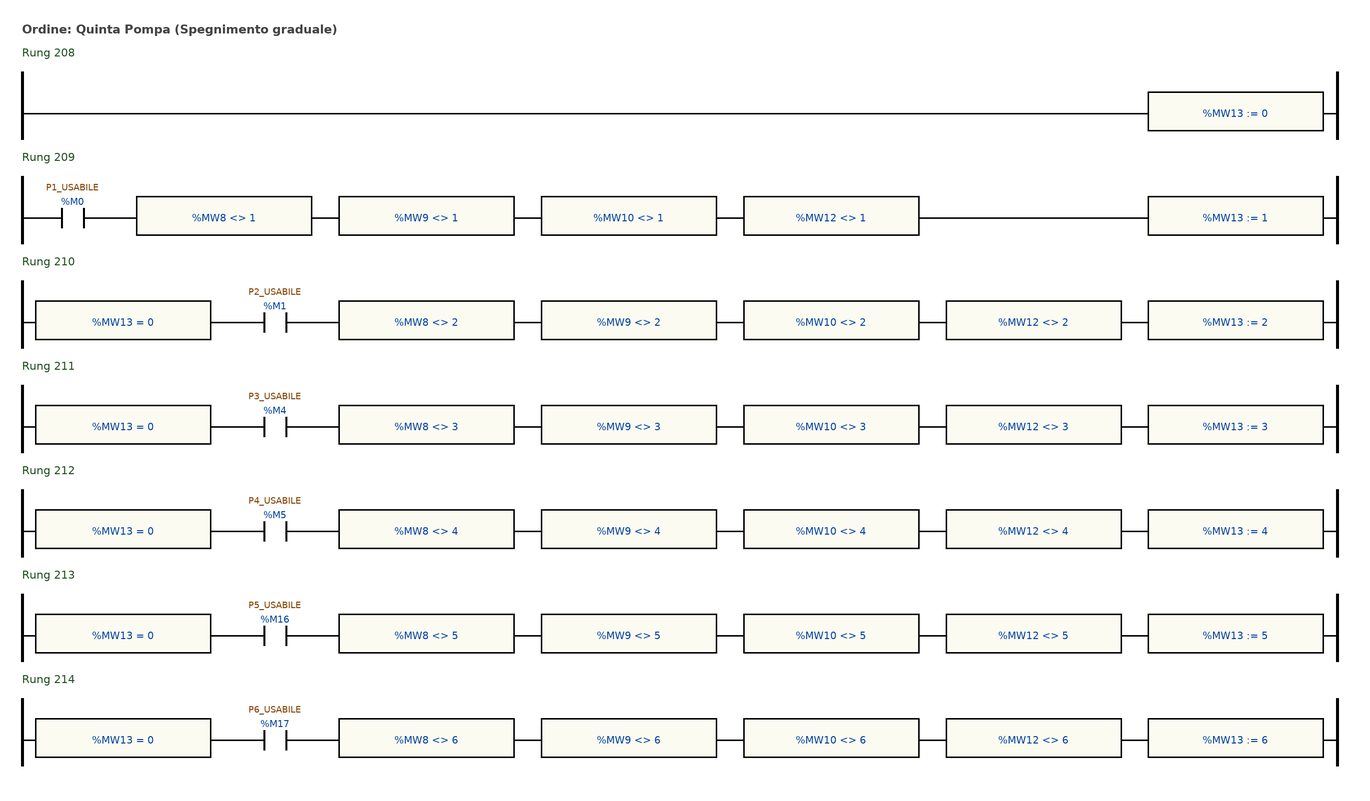

// Rung 208
  LD 1
  [ %MW13 := 0 ]          (* ORDINE_QUINTA_POMPA *)
  // as ST:
  //   ORDINE_QUINTA_POMPA := 0;

// Rung 209
  LD %M0                  (* P1_USABILE *)
  AND [ %MW8 <> 1 ]       (* ORDINE_PRIMA_POMPA *)
  AND [ %MW9 <> 1 ]       (* ORDINE_SECONDA_POMPA *)
  AND [ %MW10 <> 1 ]      (* ORDINE_TERZA_POMPA *)
  AND [ %MW12 <> 1 ]      (* ORDINE_QUARTA_POMPA *)
  [ %MW13 := 1 ]          (* ORDINE_QUINTA_POMPA *)
  // as ST:
  //   IF P1_USABILE AND ORDINE_PRIMA_POMPA <> 1 AND ORDINE_SECONDA_POMPA <> 1 AND ORDINE_TERZA_POMPA <> 1 AND ORDINE_QUARTA_POMPA <> 1 THEN ORDINE_QUINTA_POMPA := 1; END_IF;

// Rung 210
  LD [ %MW13 = 0 ]        (* ORDINE_QUINTA_POMPA *)
  AND %M1                 (* P2_USABILE *)
  AND [ %MW8 <> 2 ]       (* ORDINE_PRIMA_POMPA *)
  AND [ %MW9 <> 2 ]       (* ORDINE_SECONDA_POMPA *)
  AND [ %MW10 <> 2 ]      (* ORDINE_TERZA_POMPA *)
  AND [ %MW12 <> 2 ]      (* ORDINE_QUARTA_POMPA *)
  [ %MW13 := 2 ]          (* ORDINE_QUINTA_POMPA *)
  // as ST:
  //   IF ORDINE_QUINTA_POMPA = 0 AND P2_USABILE AND ORDINE_PRIMA_POMPA <> 2 AND ORDINE_SECONDA_POMPA <> 2 AND ORDINE_TERZA_POMPA <> 2 AND ORDINE_QUARTA_POMPA <> 2 THEN ORDINE_QUINTA_POMPA := 2; END_IF;

// Rung 211
  LD [ %MW13 = 0 ]        (* ORDINE_QUINTA_POMPA *)
  AND %M4                 (* P3_USABILE *)
  AND [ %MW8 <> 3 ]       (* ORDINE_PRIMA_POMPA *)
  AND [ %MW9 <> 3 ]       (* ORDINE_SECONDA_POMPA *)
  AND [ %MW10 <> 3 ]      (* ORDINE_TERZA_POMPA *)
  AND [ %MW12 <> 3 ]      (* ORDINE_QUARTA_POMPA *)
  [ %MW13 := 3 ]          (* ORDINE_QUINTA_POMPA *)
  // as ST:
  //   IF ORDINE_QUINTA_POMPA = 0 AND P3_USABILE AND ORDINE_PRIMA_POMPA <> 3 AND ORDINE_SECONDA_POMPA <> 3 AND ORDINE_TERZA_POMPA <> 3 AND ORDINE_QUARTA_POMPA <> 3 THEN ORDINE_QUINTA_POMPA := 3; END_IF;

// Rung 212
  LD [ %MW13 = 0 ]        (* ORDINE_QUINTA_POMPA *)
  AND %M5                 (* P4_USABILE *)
  AND [ %MW8 <> 4 ]       (* ORDINE_PRIMA_POMPA *)
  AND [ %MW9 <> 4 ]       (* ORDINE_SECONDA_POMPA *)
  AND [ %MW10 <> 4 ]      (* ORDINE_TERZA_POMPA *)
  AND [ %MW12 <> 4 ]      (* ORDINE_QUARTA_POMPA *)
  [ %MW13 := 4 ]          (* ORDINE_QUINTA_POMPA *)
  // as ST:
  //   IF ORDINE_QUINTA_POMPA = 0 AND P4_USABILE AND ORDINE_PRIMA_POMPA <> 4 AND ORDINE_SECONDA_POMPA <> 4 AND ORDINE_TERZA_POMPA <> 4 AND ORDINE_QUARTA_POMPA <> 4 THEN ORDINE_QUINTA_POMPA := 4; END_IF;

// Rung 213
  LD [ %MW13 = 0 ]        (* ORDINE_QUINTA_POMPA *)
  AND %M16                (* P5_USABILE *)
  AND [ %MW8 <> 5 ]       (* ORDINE_PRIMA_POMPA *)
  AND [ %MW9 <> 5 ]       (* ORDINE_SECONDA_POMPA *)
  AND [ %MW10 <> 5 ]      (* ORDINE_TERZA_POMPA *)
  AND [ %MW12 <> 5 ]      (* ORDINE_QUARTA_POMPA *)
  [ %MW13 := 5 ]          (* ORDINE_QUINTA_POMPA *)
  // as ST:
  //   IF ORDINE_QUINTA_POMPA = 0 AND P5_USABILE AND ORDINE_PRIMA_POMPA <> 5 AND ORDINE_SECONDA_POMPA <> 5 AND ORDINE_TERZA_POMPA <> 5 AND ORDINE_QUARTA_POMPA <> 5 THEN ORDINE_QUINTA_POMPA := 5; END_IF;

// Rung 214
  LD [ %MW13 = 0 ]        (* ORDINE_QUINTA_POMPA *)
  AND %M17                (* P6_USABILE *)
  AND [ %MW8 <> 6 ]       (* ORDINE_PRIMA_POMPA *)
  AND [ %MW9 <> 6 ]       (* ORDINE_SECONDA_POMPA *)
  AND [ %MW10 <> 6 ]      (* ORDINE_TERZA_POMPA *)
  AND [ %MW12 <> 6 ]      (* ORDINE_QUARTA_POMPA *)
  [ %MW13 := 6 ]          (* ORDINE_QUINTA_POMPA *)
  // as ST:
  //   IF ORDINE_QUINTA_POMPA = 0 AND P6_USABILE AND ORDINE_PRIMA_POMPA <> 6 AND ORDINE_SECONDA_POMPA <> 6 AND ORDINE_TERZA_POMPA <> 6 AND ORDINE_QUARTA_POMPA <> 6 THEN ORDINE_QUINTA_POMPA := 6; END_IF;

Subroutine Comanda: Quarta Pompa (Spegnimento graduale)
  (* SectionNumber=30, Number=28 *)

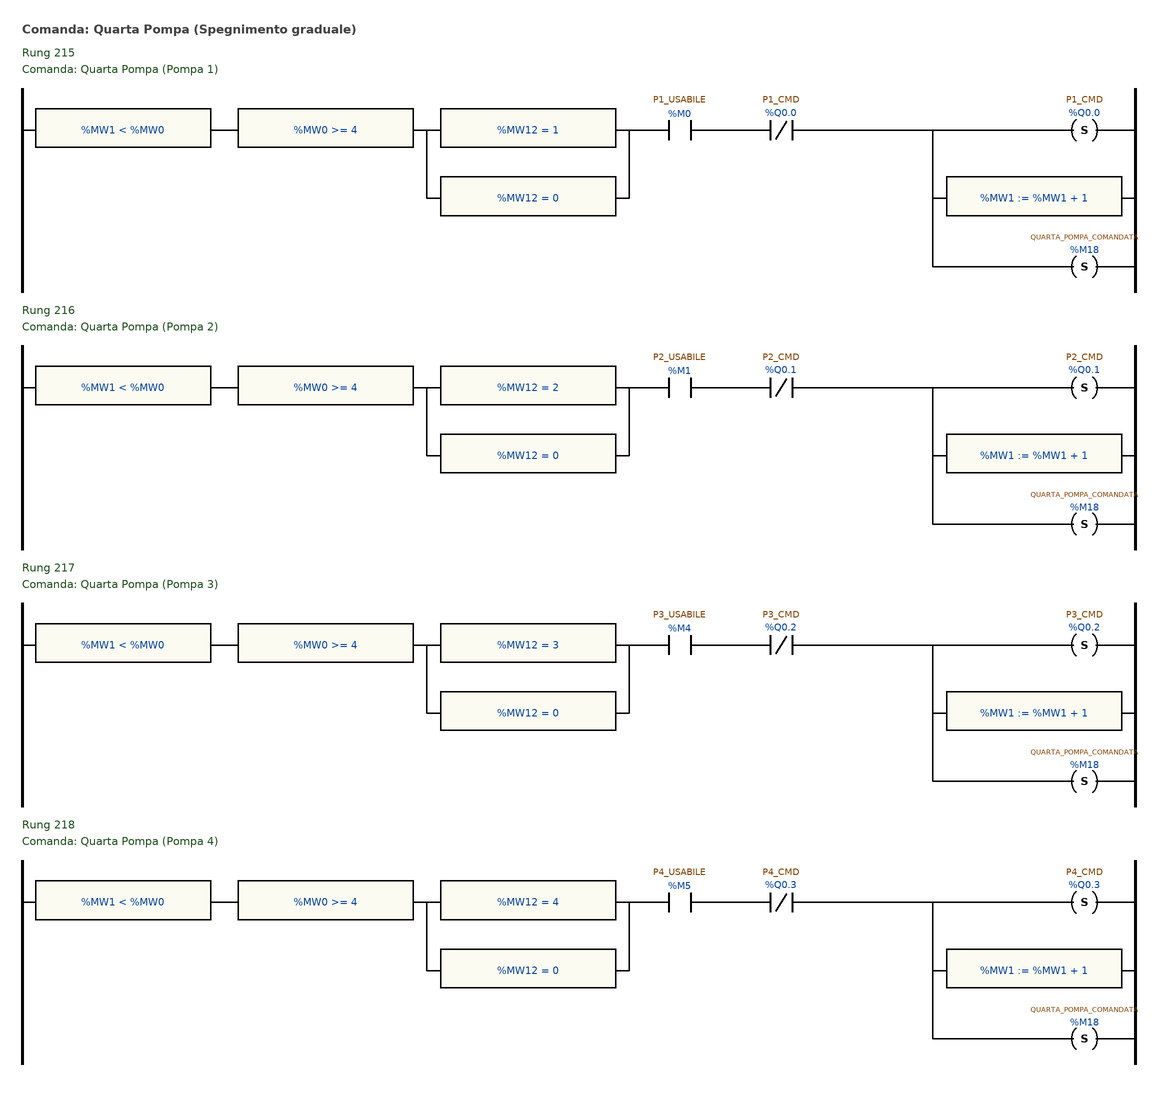

// Rung 215
// Comanda: Quarta Pompa (Pompa 1)
  LD [ %MW1 < %MW0 ]      (* NUM_POMPE_COMANDATE, NUM_POMPE_DA_COMANDARE *)
  AND [ %MW0 >= 4 ]       (* NUM_POMPE_DA_COMANDARE *)
  AND( [ %MW12 = 1 ]      (* ORDINE_QUARTA_POMPA *)
  OR [ %MW12 = 0 ]        (* ORDINE_QUARTA_POMPA *)
  )
  AND %M0                 (* P1_USABILE *)
  ANDN %Q0.0              (* P1_CMD *)
  S %Q0.0                 (* P1_CMD *)
  [ %MW1 := %MW1 + 1 ]    (* NUM_POMPE_COMANDATE, NUM_POMPE_COMANDATE *)
  S %M18                  (* QUARTA_POMPA_COMANDATA *)
  // as ST:
  //   _t1 := NUM_POMPE_COMANDATE < NUM_POMPE_DA_COMANDARE AND NUM_POMPE_DA_COMANDARE >= 4 AND (ORDINE_QUARTA_POMPA = 1 OR ORDINE_QUARTA_POMPA = 0) AND P1_USABILE AND NOT P1_CMD;
  //   IF _t1 THEN P1_CMD := TRUE; END_IF;
  //   IF _t1 THEN NUM_POMPE_COMANDATE := NUM_POMPE_COMANDATE + 1; END_IF;
  //   IF _t1 THEN QUARTA_POMPA_COMANDATA := TRUE; END_IF;

// Rung 216
// Comanda: Quarta Pompa (Pompa 2)
  LD [ %MW1 < %MW0 ]      (* NUM_POMPE_COMANDATE, NUM_POMPE_DA_COMANDARE *)
  AND [ %MW0 >= 4 ]       (* NUM_POMPE_DA_COMANDARE *)
  AND( [ %MW12 = 2 ]      (* ORDINE_QUARTA_POMPA *)
  OR [ %MW12 = 0 ]        (* ORDINE_QUARTA_POMPA *)
  )
  AND %M1                 (* P2_USABILE *)
  ANDN %Q0.1              (* P2_CMD *)
  S %Q0.1                 (* P2_CMD *)
  [ %MW1 := %MW1 + 1 ]    (* NUM_POMPE_COMANDATE, NUM_POMPE_COMANDATE *)
  S %M18                  (* QUARTA_POMPA_COMANDATA *)
  // as ST:
  //   _t1 := NUM_POMPE_COMANDATE < NUM_POMPE_DA_COMANDARE AND NUM_POMPE_DA_COMANDARE >= 4 AND (ORDINE_QUARTA_POMPA = 2 OR ORDINE_QUARTA_POMPA = 0) AND P2_USABILE AND NOT P2_CMD;
  //   IF _t1 THEN P2_CMD := TRUE; END_IF;
  //   IF _t1 THEN NUM_POMPE_COMANDATE := NUM_POMPE_COMANDATE + 1; END_IF;
  //   IF _t1 THEN QUARTA_POMPA_COMANDATA := TRUE; END_IF;

// Rung 217
// Comanda: Quarta Pompa (Pompa 3)
  LD [ %MW1 < %MW0 ]      (* NUM_POMPE_COMANDATE, NUM_POMPE_DA_COMANDARE *)
  AND [ %MW0 >= 4 ]       (* NUM_POMPE_DA_COMANDARE *)
  AND( [ %MW12 = 3 ]      (* ORDINE_QUARTA_POMPA *)
  OR [ %MW12 = 0 ]        (* ORDINE_QUARTA_POMPA *)
  )
  AND %M4                 (* P3_USABILE *)
  ANDN %Q0.2              (* P3_CMD *)
  S %Q0.2                 (* P3_CMD *)
  [ %MW1 := %MW1 + 1 ]    (* NUM_POMPE_COMANDATE, NUM_POMPE_COMANDATE *)
  S %M18                  (* QUARTA_POMPA_COMANDATA *)
  // as ST:
  //   _t1 := NUM_POMPE_COMANDATE < NUM_POMPE_DA_COMANDARE AND NUM_POMPE_DA_COMANDARE >= 4 AND (ORDINE_QUARTA_POMPA = 3 OR ORDINE_QUARTA_POMPA = 0) AND P3_USABILE AND NOT P3_CMD;
  //   IF _t1 THEN P3_CMD := TRUE; END_IF;
  //   IF _t1 THEN NUM_POMPE_COMANDATE := NUM_POMPE_COMANDATE + 1; END_IF;
  //   IF _t1 THEN QUARTA_POMPA_COMANDATA := TRUE; END_IF;

// Rung 218
// Comanda: Quarta Pompa (Pompa 4)
  LD [ %MW1 < %MW0 ]      (* NUM_POMPE_COMANDATE, NUM_POMPE_DA_COMANDARE *)
  AND [ %MW0 >= 4 ]       (* NUM_POMPE_DA_COMANDARE *)
  AND( [ %MW12 = 4 ]      (* ORDINE_QUARTA_POMPA *)
  OR [ %MW12 = 0 ]        (* ORDINE_QUARTA_POMPA *)
  )
  AND %M5                 (* P4_USABILE *)
  ANDN %Q0.3              (* P4_CMD *)
  S %Q0.3                 (* P4_CMD *)
  [ %MW1 := %MW1 + 1 ]    (* NUM_POMPE_COMANDATE, NUM_POMPE_COMANDATE *)
  S %M18                  (* QUARTA_POMPA_COMANDATA *)
  // as ST:
  //   _t1 := NUM_POMPE_COMANDATE < NUM_POMPE_DA_COMANDARE AND NUM_POMPE_DA_COMANDARE >= 4 AND (ORDINE_QUARTA_POMPA = 4 OR ORDINE_QUARTA_POMPA = 0) AND P4_USABILE AND NOT P4_CMD;
  //   IF _t1 THEN P4_CMD := TRUE; END_IF;
  //   IF _t1 THEN NUM_POMPE_COMANDATE := NUM_POMPE_COMANDATE + 1; END_IF;
  //   IF _t1 THEN QUARTA_POMPA_COMANDATA := TRUE; END_IF;

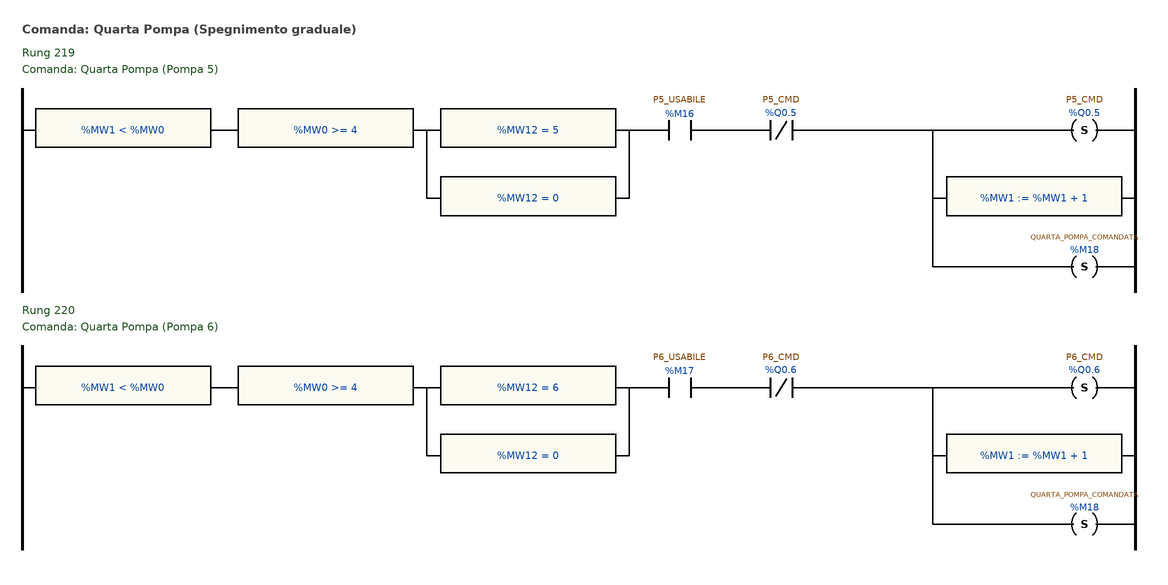

// Rung 219
// Comanda: Quarta Pompa (Pompa 5)
  LD [ %MW1 < %MW0 ]      (* NUM_POMPE_COMANDATE, NUM_POMPE_DA_COMANDARE *)
  AND [ %MW0 >= 4 ]       (* NUM_POMPE_DA_COMANDARE *)
  AND( [ %MW12 = 5 ]      (* ORDINE_QUARTA_POMPA *)
  OR [ %MW12 = 0 ]        (* ORDINE_QUARTA_POMPA *)
  )
  AND %M16                (* P5_USABILE *)
  ANDN %Q0.5              (* P5_CMD *)
  S %Q0.5                 (* P5_CMD *)
  [ %MW1 := %MW1 + 1 ]    (* NUM_POMPE_COMANDATE, NUM_POMPE_COMANDATE *)
  S %M18                  (* QUARTA_POMPA_COMANDATA *)
  // as ST:
  //   _t1 := NUM_POMPE_COMANDATE < NUM_POMPE_DA_COMANDARE AND NUM_POMPE_DA_COMANDARE >= 4 AND (ORDINE_QUARTA_POMPA = 5 OR ORDINE_QUARTA_POMPA = 0) AND P5_USABILE AND NOT P5_CMD;
  //   IF _t1 THEN P5_CMD := TRUE; END_IF;
  //   IF _t1 THEN NUM_POMPE_COMANDATE := NUM_POMPE_COMANDATE + 1; END_IF;
  //   IF _t1 THEN QUARTA_POMPA_COMANDATA := TRUE; END_IF;

// Rung 220
// Comanda: Quarta Pompa (Pompa 6)
  LD [ %MW1 < %MW0 ]      (* NUM_POMPE_COMANDATE, NUM_POMPE_DA_COMANDARE *)
  AND [ %MW0 >= 4 ]       (* NUM_POMPE_DA_COMANDARE *)
  AND( [ %MW12 = 6 ]      (* ORDINE_QUARTA_POMPA *)
  OR [ %MW12 = 0 ]        (* ORDINE_QUARTA_POMPA *)
  )
  AND %M17                (* P6_USABILE *)
  ANDN %Q0.6              (* P6_CMD *)
  S %Q0.6                 (* P6_CMD *)
  [ %MW1 := %MW1 + 1 ]    (* NUM_POMPE_COMANDATE, NUM_POMPE_COMANDATE *)
  S %M18                  (* QUARTA_POMPA_COMANDATA *)
  // as ST:
  //   _t1 := NUM_POMPE_COMANDATE < NUM_POMPE_DA_COMANDARE AND NUM_POMPE_DA_COMANDARE >= 4 AND (ORDINE_QUARTA_POMPA = 6 OR ORDINE_QUARTA_POMPA = 0) AND P6_USABILE AND NOT P6_CMD;
  //   IF _t1 THEN P6_CMD := TRUE; END_IF;
  //   IF _t1 THEN NUM_POMPE_COMANDATE := NUM_POMPE_COMANDATE + 1; END_IF;
  //   IF _t1 THEN QUARTA_POMPA_COMANDATA := TRUE; END_IF;

Subroutine Comanda: Quinta Pompa (Spegnimento graduale)
  (* SectionNumber=31, Number=29 *)

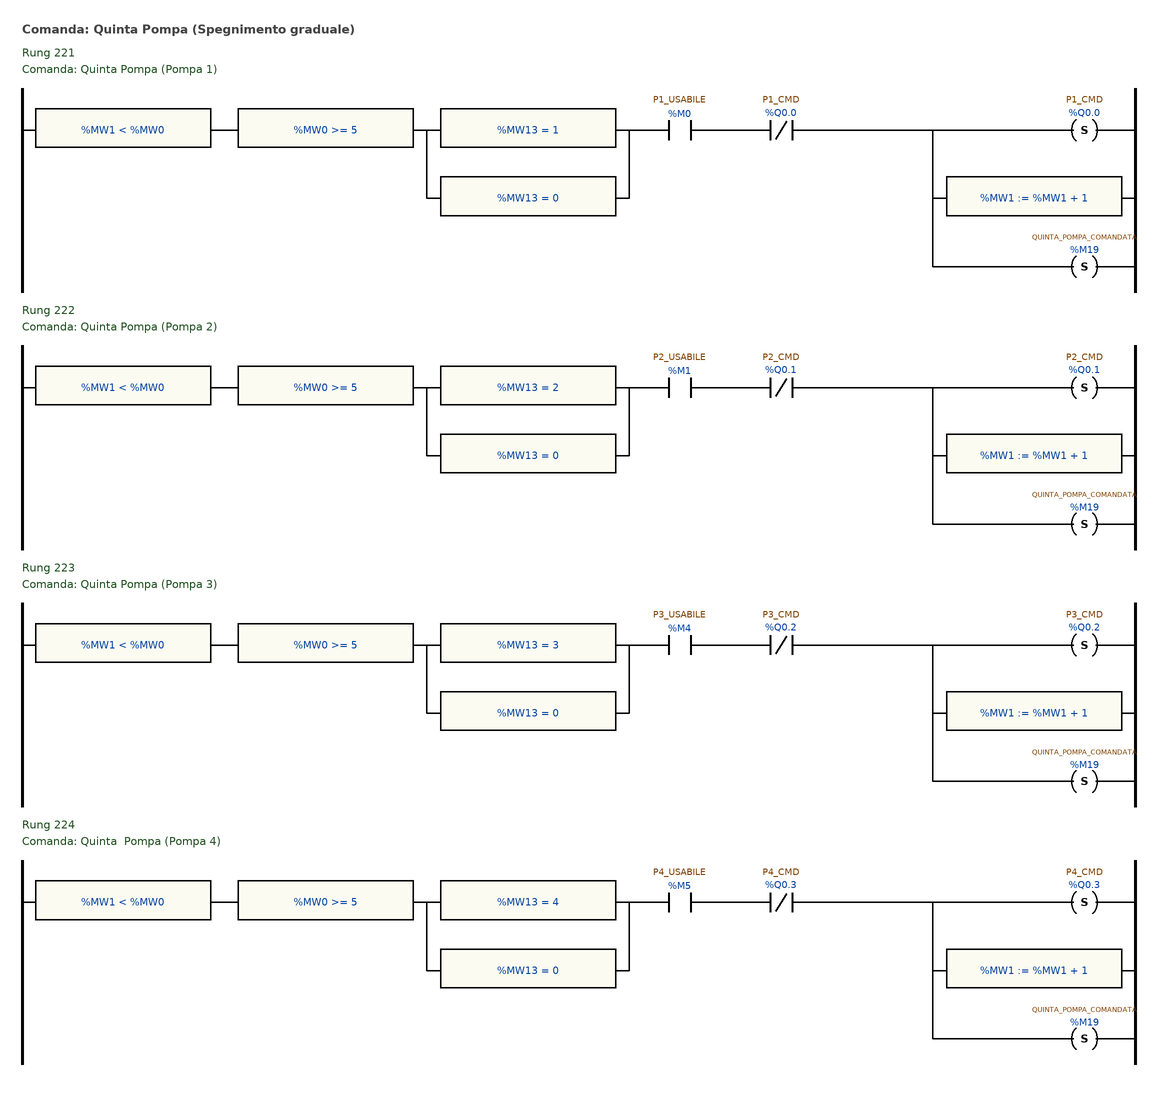

// Rung 221
// Comanda: Quinta Pompa (Pompa 1)
  LD [ %MW1 < %MW0 ]      (* NUM_POMPE_COMANDATE, NUM_POMPE_DA_COMANDARE *)
  AND [ %MW0 >= 5 ]       (* NUM_POMPE_DA_COMANDARE *)
  AND( [ %MW13 = 1 ]      (* ORDINE_QUINTA_POMPA *)
  OR [ %MW13 = 0 ]        (* ORDINE_QUINTA_POMPA *)
  )
  AND %M0                 (* P1_USABILE *)
  ANDN %Q0.0              (* P1_CMD *)
  S %Q0.0                 (* P1_CMD *)
  [ %MW1 := %MW1 + 1 ]    (* NUM_POMPE_COMANDATE, NUM_POMPE_COMANDATE *)
  S %M19                  (* QUINTA_POMPA_COMANDATA *)
  // as ST:
  //   _t1 := NUM_POMPE_COMANDATE < NUM_POMPE_DA_COMANDARE AND NUM_POMPE_DA_COMANDARE >= 5 AND (ORDINE_QUINTA_POMPA = 1 OR ORDINE_QUINTA_POMPA = 0) AND P1_USABILE AND NOT P1_CMD;
  //   IF _t1 THEN P1_CMD := TRUE; END_IF;
  //   IF _t1 THEN NUM_POMPE_COMANDATE := NUM_POMPE_COMANDATE + 1; END_IF;
  //   IF _t1 THEN QUINTA_POMPA_COMANDATA := TRUE; END_IF;

// Rung 222
// Comanda: Quinta Pompa (Pompa 2)
  LD [ %MW1 < %MW0 ]      (* NUM_POMPE_COMANDATE, NUM_POMPE_DA_COMANDARE *)
  AND [ %MW0 >= 5 ]       (* NUM_POMPE_DA_COMANDARE *)
  AND( [ %MW13 = 2 ]      (* ORDINE_QUINTA_POMPA *)
  OR [ %MW13 = 0 ]        (* ORDINE_QUINTA_POMPA *)
  )
  AND %M1                 (* P2_USABILE *)
  ANDN %Q0.1              (* P2_CMD *)
  S %Q0.1                 (* P2_CMD *)
  [ %MW1 := %MW1 + 1 ]    (* NUM_POMPE_COMANDATE, NUM_POMPE_COMANDATE *)
  S %M19                  (* QUINTA_POMPA_COMANDATA *)
  // as ST:
  //   _t1 := NUM_POMPE_COMANDATE < NUM_POMPE_DA_COMANDARE AND NUM_POMPE_DA_COMANDARE >= 5 AND (ORDINE_QUINTA_POMPA = 2 OR ORDINE_QUINTA_POMPA = 0) AND P2_USABILE AND NOT P2_CMD;
  //   IF _t1 THEN P2_CMD := TRUE; END_IF;
  //   IF _t1 THEN NUM_POMPE_COMANDATE := NUM_POMPE_COMANDATE + 1; END_IF;
  //   IF _t1 THEN QUINTA_POMPA_COMANDATA := TRUE; END_IF;

// Rung 223
// Comanda: Quinta Pompa (Pompa 3)
  LD [ %MW1 < %MW0 ]      (* NUM_POMPE_COMANDATE, NUM_POMPE_DA_COMANDARE *)
  AND [ %MW0 >= 5 ]       (* NUM_POMPE_DA_COMANDARE *)
  AND( [ %MW13 = 3 ]      (* ORDINE_QUINTA_POMPA *)
  OR [ %MW13 = 0 ]        (* ORDINE_QUINTA_POMPA *)
  )
  AND %M4                 (* P3_USABILE *)
  ANDN %Q0.2              (* P3_CMD *)
  S %Q0.2                 (* P3_CMD *)
  [ %MW1 := %MW1 + 1 ]    (* NUM_POMPE_COMANDATE, NUM_POMPE_COMANDATE *)
  S %M19                  (* QUINTA_POMPA_COMANDATA *)
  // as ST:
  //   _t1 := NUM_POMPE_COMANDATE < NUM_POMPE_DA_COMANDARE AND NUM_POMPE_DA_COMANDARE >= 5 AND (ORDINE_QUINTA_POMPA = 3 OR ORDINE_QUINTA_POMPA = 0) AND P3_USABILE AND NOT P3_CMD;
  //   IF _t1 THEN P3_CMD := TRUE; END_IF;
  //   IF _t1 THEN NUM_POMPE_COMANDATE := NUM_POMPE_COMANDATE + 1; END_IF;
  //   IF _t1 THEN QUINTA_POMPA_COMANDATA := TRUE; END_IF;

// Rung 224
// Comanda: Quinta  Pompa (Pompa 4)
  LD [ %MW1 < %MW0 ]      (* NUM_POMPE_COMANDATE, NUM_POMPE_DA_COMANDARE *)
  AND [ %MW0 >= 5 ]       (* NUM_POMPE_DA_COMANDARE *)
  AND( [ %MW13 = 4 ]      (* ORDINE_QUINTA_POMPA *)
  OR [ %MW13 = 0 ]        (* ORDINE_QUINTA_POMPA *)
  )
  AND %M5                 (* P4_USABILE *)
  ANDN %Q0.3              (* P4_CMD *)
  S %Q0.3                 (* P4_CMD *)
  [ %MW1 := %MW1 + 1 ]    (* NUM_POMPE_COMANDATE, NUM_POMPE_COMANDATE *)
  S %M19                  (* QUINTA_POMPA_COMANDATA *)
  // as ST:
  //   _t1 := NUM_POMPE_COMANDATE < NUM_POMPE_DA_COMANDARE AND NUM_POMPE_DA_COMANDARE >= 5 AND (ORDINE_QUINTA_POMPA = 4 OR ORDINE_QUINTA_POMPA = 0) AND P4_USABILE AND NOT P4_CMD;
  //   IF _t1 THEN P4_CMD := TRUE; END_IF;
  //   IF _t1 THEN NUM_POMPE_COMANDATE := NUM_POMPE_COMANDATE + 1; END_IF;
  //   IF _t1 THEN QUINTA_POMPA_COMANDATA := TRUE; END_IF;

